				IF F_ChkSettingLimit(stControlSettingIn.nInputNumber, TO_LREAL(stControlSettingIn.fInputFloat), stSettings[nRowIndex], stInfo => stInfo) THEN
					IF stSettings[nRowIndex].eDataType = E_DataType.eDataType_bool THEN
						F_TrackSettingChangesB(stControlSettingIn.bInputBool, stSettings[nRowIndex], sChanges);
					ELSIF stSettings[nRowIndex].eDataType = E_DataType.eDataType_int THEN
						F_TrackSettingChangesI(stControlSettingIn.nInputNumber, stSettings[nRowIndex], sChanges);
					ELSIF stSettings[nRowIndex].eDataType = E_DataType.eDataType_lreal THEN
						F_TrackSettingChangesF(stControlSettingIn.fInputFloat, stSettings[nRowIndex], sChanges);
					ELSIF stSettings[nRowIndex].eDataType = E_DataType.eDataType_wstring THEN
						F_TrackSettingChangesWs(stControlSettingIn.wsInputString, stSettings[nRowIndex], sChanges);
					ELSIF stSettings[nRowIndex].eDataType = E_DataType.eDataType_time_ms THEN
						F_TrackSettingChangesT(TO_TIME(stControlSettingIn.nInputNumber), stSettings[nRowIndex], sChanges);
					ELSIF stSettings[nRowIndex].eDataType = E_DataType.eDataType_time_s THEN
						F_TrackSettingChangesT(TO_TIME((stControlSettingIn.fInputFloat) * 1000), stSettings[nRowIndex], sChanges);
					ELSIF stSettings[nRowIndex].eDataType = E_DataType.eDataType_time_m THEN
						F_TrackSettingChangesT(TO_TIME((stControlSettingIn.fInputFloat) * 60000), stSettings[nRowIndex], sChanges);
					ELSIF stSettings[nRowIndex].eDataType = E_DataType.eDataType_time_h THEN
						F_TrackSettingChangesT(TO_TIME((stControlSettingIn.fInputFloat) * 360000), stSettings[nRowIndex], sChanges);
					END_IF
				ELSE
					tofInfo.IN := TRUE;
				END_IF
				
			3: // min > user level admin
				IF (eUserLevel < E_User_Level.eUser_Level_Admin) 
					OR ((stSettings[nRowIndex].eUserLevel = E_User_Level.eUser_Level_Programmer) AND (eUserLevel <> E_User_Level.eUser_Level_Programmer))
				THEN
					tofInfo.IN :=	TRUE;
					stInfo.wsName := "incorrect user level";
					stInfo.wsNameId := "incorrectuserlevel";
				ELSE
					stSettings[nRowIndex].fValueMin := stControlSettingIn.fInputFloat;
				END_IF
				
			4: // max > user level admin
				IF (eUserLevel < E_User_Level.eUser_Level_Admin) 
					OR ((stSettings[nRowIndex].eUserLevel = E_User_Level.eUser_Level_Programmer) AND (eUserLevel <> E_User_Level.eUser_Level_Programmer))
				THEN
					tofInfo.IN :=	TRUE;
					stInfo.wsName := "incorrect user level";
					stInfo.wsNameId := "incorrectuserlevel";
				ELSE
					stSettings[nRowIndex].fValueMax := stControlSettingIn.fInputFloat;
				END_IF
				
			5: // unit only write by programmer
				;
					
			6: // user level admin
				IF (eUserLevel < E_User_Level.eUser_Level_Admin) 
					OR ((stSettings[nRowIndex].eUserLevel = E_User_Level.eUser_Level_Programmer) AND (eUserLevel <> E_User_Level.eUser_Level_Programmer))
				THEN
					tofInfo.IN :=	TRUE;
					stInfo.wsName := "incorrect user level";
					stInfo.wsNameId := "incorrectuserlevel";
				ELSE
					IF (stControlSettingIn.eUserLevel = E_User_Level.eUser_Level_Programmer) AND (eUserLevel < E_User_Level.eUser_Level_Programmer) THEN
						tofInfo.IN :=	TRUE;
						stInfo.wsName := "incorrect user level";
						stInfo.wsNameId := "incorrectuserlevel";						
					ELSE
						stSettings[nRowIndex].eUserLevel := stControlSettingIn.eUserLevel;
					END_IF	
				END_IF
				
			7: // type only write by programmer
				;
				
			8: // recipe level manager
				IF (eUserLevel < E_User_Level.eUser_Level_Manager) 
					OR ((stSettings[nRowIndex].eUserLevel = E_User_Level.eUser_Level_Programmer) AND (eUserLevel <> E_User_Level.eUser_Level_Programmer))
				THEN
					tofInfo.IN :=	TRUE;
					stInfo.wsName := "incorrect user level";
					stInfo.wsNameId := "incorrectuserlevel";
				ELSE
					stSettings[nRowIndex].eRecipeMode := stControlSettingIn.eRecipeMode;
				END_IF 				
		END_CASE
	END_IF
END_IF

tofInfo.PT := T#2S;
tofInfo();
tofInfo.IN := FALSE;
		
stControlSettingOut.bVisibleInfo := tofInfo.Q;
stControlSettingOut.stInfo := stInfo;

END_FUNCTION_BLOCK

// ---- POUs/System/Utilities/Functions/F_ColorToStringHexColor.TcPOU
FUNCTION F_ColorToStringHexColor : STRING
VAR_INPUT
	color : UDINT;
END_VAR

IF color = STATICS.stColor.None THEN
	F_ColorToStringHexColor := STATICS.stColor.NoneString;
ELSIF color = STATICS.stColor.Transparent THEN
	F_ColorToStringHexColor := STATICS.stColor.TransparentString;	
ELSIF color = STATICS.stColor.Theme THEN
	F_ColorToStringHexColor := STATICS.stColor.ThemeString;
ELSE
	F_ColorToStringHexColor  := Concat(
								'#',
								Delete(
									DWORD_TO_HEXSTR(
											color,
											8,
											FALSE)
									,2
									,1));//#hexadecimal
END_IF

END_FUNCTION

// ---- POUs/HMI/Utilities/Validation/F_ChkSettingUserLevel.TcPOU
FUNCTION F_ChkSettingUserLevel : BOOL
VAR_INPUT
	eLevel		: E_User_Level;
END_VAR
VAR_IN_OUT
	stSetting 	: ST_Data_Item;
END_VAR
VAR_OUTPUT
	stInfo 		: ST_Text;
END_VAR

F_ChkSettingUserLevel := FALSE;

IF (eUserLevel < stSetting.eUserLevel) THEN
	stInfo.wsName := "incorrect user level";
	stInfo.wsNameId := "incorrectuserlevel";
	RETURN;
END_IF

IF(stSetting.eDataType = E_DataType.eDataType_None)	THEN
	stInfo.wsName := "incorrect type";
	stInfo.wsNameId := "incorrecttype";
	RETURN;					
END_IF

F_ChkSettingUserLevel := TRUE;

END_FUNCTION

// ---- POUs/HMI/Utilities/Validation/F_ChkSettingLimit.TcPOU
FUNCTION F_ChkSettingLimit : BOOL
VAR_INPUT
	nValue		: INT;
	fValue		: LREAL;
END_VAR
VAR_IN_OUT
	stSetting 	: ST_Data_Item;
END_VAR
VAR_OUTPUT
	stInfo 		: ST_Text;
END_VAR

CASE stSetting.eDataType OF
	E_DataType.eDataType_int,
	E_DataType.eDataType_time_ms:
		F_ChkSettingLimit := F_ChkSettingLimitN(nValue, stSetting, stInfo => stInfo);
ELSE
		F_ChkSettingLimit := F_ChkSettingLimitF(fValue, stSetting, stInfo => stInfo);
END_CASE

END_FUNCTION

// ---- POUs/HMI/Utilities/Validation/F_ChkSettingLimitN.TcPOU
FUNCTION F_ChkSettingLimitN : BOOL
VAR_IN_OUT
	nValue		: INT;
	stSetting 	: ST_Data_Item;
END_VAR
VAR_OUTPUT
	stInfo 		: ST_Text;
END_VAR

F_ChkSettingLimitN := FALSE;

IF (stSetting.eDataType = E_DataType.eDataType_int) AND nValue > stSetting.fValueMax THEN
	stInfo.wsName := "input to high";
	stInfo.wsNameId := "inputtohigh";
	RETURN;
END_IF

IF (stSetting.eDataType = E_DataType.eDataType_int) AND nValue < stSetting.fValueMin THEN
	stInfo.wsName := "input to low";
	stInfo.wsNameId := "inputtolow";
	RETURN;
END_IF

IF (stSetting.eDataType = E_DataType.eDataType_time_ms) AND nValue > stSetting.fValueMax THEN
	stInfo.wsName := "input to high";
	stInfo.wsNameId := "inputtohigh";
	RETURN;
END_IF

IF (stSetting.eDataType = E_DataType.eDataType_time_ms) AND nValue < stSetting.fValueMin THEN
	stInfo.wsName := "input to low";
	stInfo.wsNameId := "inputtolow";
	RETURN;
END_IF

F_ChkSettingLimitN := TRUE;

END_FUNCTION

// ---- POUs/HMI/Utilities/Validation/F_ChkSettingLimitF.TcPOU
FUNCTION F_ChkSettingLimitF : BOOL
VAR_IN_OUT
	fValue		: LREAL;
	stSetting 	: ST_Data_Item;
END_VAR
VAR_OUTPUT
	stInfo 		: ST_Text;
END_VAR

F_ChkSettingLimitF := FALSE;

IF (stSetting.eDataType = E_DataType.eDataType_lreal) AND fValue > stSetting.fValueMax THEN
	stInfo.wsName := "input to high";
	stInfo.wsNameId := "inputtohigh";
	RETURN;
END_IF

IF (stSetting.eDataType = E_DataType.eDataType_lreal) AND fValue < stSetting.fValueMin THEN
	stInfo.wsName := "input to low";
	stInfo.wsNameId := "inputtolow";
	RETURN;
END_IF

IF (stSetting.eDataType = E_DataType.eDataType_time_s) AND fValue > stSetting.fValueMax THEN
	stInfo.wsName := "input to high";
	stInfo.wsNameId := "inputtohigh";
	RETURN;
END_IF

IF (stSetting.eDataType = E_DataType.eDataType_time_s) AND fValue < stSetting.fValueMin THEN
	stInfo.wsName := "input to low";
	stInfo.wsNameId := "inputtolow";
	RETURN;
END_IF

IF (stSetting.eDataType = E_DataType.eDataType_time_m) AND fValue > stSetting.fValueMax THEN
	stInfo.wsName := "input to high";
	stInfo.wsNameId := "inputtohigh";
	RETURN;
END_IF

IF (stSetting.eDataType = E_DataType.eDataType_time_m) AND fValue < stSetting.fValueMin THEN
	stInfo.wsName := "input to low";
	stInfo.wsNameId := "inputtolow";
	RETURN;
END_IF

IF (stSetting.eDataType = E_DataType.eDataType_time_h) AND fValue > stSetting.fValueMax THEN
	stInfo.wsName := "input to high";
	stInfo.wsNameId := "inputtohigh";
	RETURN;
END_IF

IF (stSetting.eDataType = E_DataType.eDataType_time_h) AND fValue < stSetting.fValueMin THEN
	stInfo.wsName := "input to low";
	stInfo.wsNameId := "inputtolow";
	RETURN;
END_IF

F_ChkSettingLimitF := TRUE;

END_FUNCTION

// ---- POUs/HMI/Utilities/Tracking/F_TrackSettingChangesB.TcPOU
FUNCTION F_TrackSettingChangesB : BOOL
VAR_INPUT
	bValue		: BOOL;
END_VAR
VAR_IN_OUT
	stSetting	: ST_Data_Item;
	sChanges	: STRING;
END_VAR

IF stSetting.bValue <> bValue THEN
	sChanges := Concat7(sChanges, '$N ', WSTRING_TO_STRING(stSetting.stName.wsName), ' ', TO_STRING(stSetting.bValue), ' -> ', TO_STRING(bValue));
END_IF

stSetting.bValue := bValue;
F_TrackSettingChangesB := TRUE;

END_FUNCTION

// ---- POUs/HMI/Utilities/Tracking/F_TrackSettingChangesI.TcPOU
FUNCTION F_TrackSettingChangesI : BOOL
VAR_INPUT
	nValue		: INT;
END_VAR
VAR_IN_OUT
	stSetting	: ST_Data_Item;
	sChanges	: STRING;
END_VAR

IF stSetting.nValue <> nValue THEN
	sChanges := Concat7(sChanges, '$N ', WSTRING_TO_STRING(stSetting.stName.wsName), ' ', TO_STRING(stSetting.nValue), ' -> ', TO_STRING(nValue));
END_IF

stSetting.nValue := nValue;
F_TrackSettingChangesI := TRUE;

END_FUNCTION

// ---- POUs/HMI/Utilities/Tracking/F_TrackSettingChangesF.TcPOU
FUNCTION F_TrackSettingChangesF : BOOL
VAR_INPUT
	fValue		: REAL;
END_VAR
VAR_IN_OUT
	stSetting	: ST_Data_Item;
	sChanges	: STRING;
END_VAR

IF stSetting.fValue <> fValue THEN
	sChanges := Concat7(sChanges, '$N ', WSTRING_TO_STRING(stSetting.stName.wsName), ' ', TO_STRING(stSetting.fValue), ' -> ', TO_STRING(fValue));
END_IF

stSetting.fValue := fValue;
F_TrackSettingChangesF := TRUE;

END_FUNCTION

// ---- POUs/HMI/Utilities/Tracking/F_TrackSettingChangesWs.TcPOU
FUNCTION F_TrackSettingChangesWs : BOOL
VAR_INPUT
	sValue		: WSTRING;
END_VAR
VAR_IN_OUT
	stSetting	: ST_Data_Item;
	sChanges	: STRING;
END_VAR

IF stSetting.sValue <> sValue THEN
	sChanges := Concat7(sChanges, '$N ', WSTRING_TO_STRING(stSetting.stName.wsName), ' ', TO_STRING(stSetting.sValue), ' -> ', TO_STRING(sValue));
END_IF

stSetting.sValue := sValue;
F_TrackSettingChangesWs := TRUE;

END_FUNCTION

// ---- POUs/HMI/Utilities/Tracking/F_TrackSettingChangesT.TcPOU
FUNCTION F_TrackSettingChangesT : BOOL
VAR_INPUT
	tValue		: TIME;
END_VAR
VAR_IN_OUT
	stSetting	: ST_Data_Item;
	sChanges	: STRING;
END_VAR

IF stSetting.tValue <> tValue THEN
	sChanges := Concat7(sChanges, '$N ', WSTRING_TO_STRING(stSetting.stName.wsName), ' ', TO_STRING(stSetting.tValue), ' -> ', TO_STRING(tValue));
END_IF

stSetting.tValue := tValue;
F_TrackSettingChangesT := TRUE;

END_FUNCTION

// ---- POUs/HMI/Utilities/FB_MonitoringHandling.TcPOU
FUNCTION_BLOCK FB_MonitoringHandling
VAR_INPUT
	nDigits				: INT; //number of digits after decimal point
END_VAR
VAR_IN_OUT
	stMonitoring		: ARRAY[*] OF ST_Data_Item;
	stMonitoringView	: ARRAY[*] OF ST_Data_Item_String;
END_VAR
VAR_OUTPUT
	
END_VAR
VAR
	ii, nLb, nUb		: DINT;
END_VAR

// clear MonitoringView
nLb := LOWER_BOUND(stMonitoringView, 1);
nUb := UPPER_BOUND(stMonitoringView, 1);
FOR ii := nLb TO nUb DO
	MEMSET(ADR(stMonitoringView[ii]), 0, SIZEOF(stMonitoringView[ii]));
END_FOR

// write MonitoringView
nLb := MAX(nLb, LOWER_BOUND(stMonitoring, 1));
nUb := MIN(nUb, UPPER_BOUND(stMonitoring, 1));
FOR ii := nLb TO nUb DO

	stMonitoringView[ii].stGroup := stMonitoring[ii].stGroup;
	stMonitoringView[ii].stName := stMonitoring[ii].stName;
	stMonitoringView[ii].stUnit := stMonitoring[ii].stUnit;
	
	IF (stMonitoring[ii].stName.wsName = "" AND stMonitoring[ii].stName.wsNameId = "") THEN
		stMonitoringView[ii].stDataType.wsName := stMonitoringView[ii].stDataType.wsNameId :="";	
	ELSIF stMonitoring[ii].eDataType = E_DataType.eDataType_None THEN
		stMonitoringView[ii].stDataType.wsName := stMonitoringView[ii].stDataType.wsNameId :="none";	
	ELSIF stMonitoring[ii].eDataType = E_DataType.eDataType_bool THEN
		stMonitoringView[ii].stDataType.wsName := stMonitoringView[ii].stDataType.wsNameId :="bool";
	ELSIF  stMonitoring[ii].eDataType = E_DataType.eDataType_int THEN
		stMonitoringView[ii].stDataType.wsName := stMonitoringView[ii].stDataType.wsNameId :="int";
	ELSIF  stMonitoring[ii].eDataType = E_DataType.eDataType_lreal THEN
		stMonitoringView[ii].stDataType.wsName := stMonitoringView[ii].stDataType.wsNameId :="lreal";
	ELSIF  stMonitoring[ii].eDataType = E_DataType.eDataType_time_ms THEN
		stMonitoringView[ii].stDataType.wsName := stMonitoringView[ii].stDataType.wsNameId :="time_ms";
	ELSIF  stMonitoring[ii].eDataType = E_DataType.eDataType_time_s THEN
		stMonitoringView[ii].stDataType.wsName := stMonitoringView[ii].stDataType.wsNameId :="time_s";		
	ELSIF  stMonitoring[ii].eDataType = E_DataType.eDataType_wstring THEN
		stMonitoringView[ii].stDataType.wsName := stMonitoringView[ii].stDataType.wsNameId :="wstring";
	END_IF
	
	IF (stMonitoring[ii].stName.wsName = "" AND stMonitoring[ii].stName.wsNameId = "") THEN
		stMonitoringView[ii].stValue.wsName := stMonitoringView[ii].stValue.wsNameId :="";
	ELSIF stMonitoring[ii].eDataType = E_DataType.eDataType_bool THEN
		IF stMonitoring[ii].bValue THEN
			stMonitoringView[ii].stValue.wsName := stMonitoringView[ii].stValue.wsNameId :="true";
		ELSE
			stMonitoringView[ii].stValue.wsName := stMonitoringView[ii].stValue.wsNameId :="false";
		END_IF
	ELSIF stMonitoring[ii].eDataType = E_DataType.eDataType_int THEN
		stMonitoringView[ii].stValue.wsName := TO_WSTRING(stMonitoring[ii].nValue);
	ELSIF stMonitoring[ii].eDataType = E_DataType.eDataType_lreal THEN
		stMonitoringView[ii].stValue.wsName := TO_WSTRING(LREAL_TO_FMTSTR(stMonitoring[ii].fValue,nDigits,FALSE));
	ELSIF stMonitoring[ii].eDataType = E_DataType.eDataType_wstring THEN
		stMonitoringView[ii].stValue.wsName := TO_WSTRING(stMonitoring[ii].sValue);
	ELSIF stMonitoring[ii].eDataType = E_DataType.eDataType_time_ms THEN
		stMonitoringView[ii].stValue.wsName := TO_WSTRING(stMonitoring[ii].tValue);
	END_IF
END_FOR

END_FUNCTION_BLOCK

// ---- POUs/System/Utilities/Functions/F_OR_REF.TcPOU
FUNCTION F_OR_REF : BOOL
VAR_IN_OUT
	bValueRoot		: BOOL;
END_VAR
VAR_INPUT
	bValueCombine	: BOOL;
END_VAR

bValueRoot := bValueRoot OR bValueCombine;

END_FUNCTION

// ---- POUs/Plant/P_Plant.TcPOU
PROGRAM P_Plant
VAR_INPUT	
	/// - stations, modules and components -
	aIStaton			: ARRAY[0..E_Station.eStation_nMaxIdx] OF IStation;
	aIModule			: ARRAY[0..E_Module.eModule_nMaxIdx] OF IModule;
	aIComponent			: ARRAY[0..E_Component.eComponent_nMaxIdx] OF ITFComponent;
END_VAR
VAR
	bInitSettingPlant		: BOOL;
	bInitSettingProduct		: BOOL;
	bInitSettingProduction	: BOOL;
	
	// plant empty... 
	bPlantEmptyActiv	: BOOL;
	bPlantEmpty			: BOOL;
	// logger, notification handler
	ILog				: I_Logger;
	IEvent				: I_EventHandler;
	
	/// private var's
	ii					: INT;
	b1stShot			: BOOL;
	tonDelay			: TON;
	
	/// clear text info
	aSClearText			: ARRAY[0..eLanguage_maxIdx] OF T_MaxString;
	bInitCounter		: BOOL;
	
	stSettingsPlantBackup		: ARRAY[0..E_PlantSettings.ePlantSetting_nMaxIdx] OF ST_Data_Item;
	stSettingsProductBackup		: ARRAY[0..E_ProductSettings.eProductSettings_nMaxIdx] OF ST_Data_Item;
	stSettingsProductionBackup	: ARRAY[0..E_ProductionSettings.eProductionSettings_nMaxIdx] OF ST_Data_Item;
END_VAR

///
/// Plant
///

// run 
aSClearText[EN] := 'Manage settings for plant, product and production';
M_SettingsPlant();
M_SettingsProduct();
M_SettingsProduction();

aSClearText[EN] := 'Calling modules...';
FOR ii := 0 TO E_Module.eModule_nMaxIdx DO
	IF aIModule[ii] = 0 THEN
		CONTINUE;
	END_IF
	
	aIModule[ii].EmergencyStopOk := P_Safety.EmergencyStopOk;
	aIModule[ii].M_Run(); // station run is called by its module
END_FOR

aSClearText[EN] := 'Calling stations, collect infos...';
b1stShot := TRUE;
FOR ii := 0 TO E_Station.eStation_nMaxIdx DO
	IF aIStaton[ii] = 0 THEN
		CONTINUE;
	END_IF
	
	F_AND_REF_EX(stGlobalModuleInfo.bStation_All_Auto, aIStaton[ii].OpMode = E_OpMode.eOpMode_auto, b1stShot);
	F_OR_REF_EX(stGlobalModuleInfo.bStation_Any_Step, aIStaton[ii].OpMode = E_OpMode.eOpMode_step, b1stShot);
	F_OR_REF_EX(stGlobalModuleInfo.bStation_Any_Manual, aIStaton[ii].OpMode = E_OpMode.eOpMode_manual, b1stShot);
	
	F_OR_REF_EX(stGlobalModuleInfo.bStation_Any_Error, aIStaton[ii].State = E_ComponentState.eComponentState_error, b1stShot);
	F_OR_REF_EX(stGlobalModuleInfo.bStation_Any_Warning, aIStaton[ii].State = E_ComponentState.eComponentState_warning, b1stShot);
	F_OR_REF_EX(stGlobalModuleInfo.bStation_Any_Info, aIStaton[ii].State = E_ComponentState.eComponentState_info, b1stShot);
	
	F_AND_REF_EX(stGlobalModuleInfo.bStation_All_Started, (aIStaton[ii].OpMode = E_OpMode.eOpMode_auto OR aIStaton[ii].OpMode = E_OpMode.eOpMode_step) AND aIStaton[ii].RunCycle, b1stShot);
	F_AND_REF_EX(stGlobalModuleInfo.bStation_All_Stopped, aIStaton[ii].Stopped, b1stShot);
	F_AND_REF_EX(stGlobalModuleInfo.bStation_All_InHome, aIStaton[ii].InHome, b1stShot);
	F_OR_REF_EX(stGlobalModuleInfo.bStation_Any_Homing, aIStaton[ii].Homing, b1stShot);
	
	b1stShot := FALSE;
END_FOR

aSClearText[EN] := 'Calling stations, plant components...';
FOR ii := 0 TO E_Component.eComponent_nMaxIdx DO
	IF aIComponent[ii] = 0 THEN
		CONTINUE;
	END_IF
	
	aIComponent[ii].Run();
END_FOR

aSClearText[EN] := 'Calling counter, check reset...';
IF HMI.stHmi.stIn.stMain.stButton_Reset.bClick THEN
	M_Reset();
END_IF

M_Counter();

IF bPlantEmptyActiv THEN
	IEvent.Select(Tc_Events.PlantEventClass.InfoEvent)
		  .ArgSetWString(CONST.stTextListGlobal.stText_emptymodeactive.wsName)
		  .Raise();
END_IF

{attribute 'monitoring' := 'call'}
PROPERTY PUBLIC CarrierColumnDistance : LREAL
GET
CarrierColumnDistance := stSettings.stProduct_Settings[E_ProductSettings.eProductSettings_CarrierColumnDistance].fValue;
END_GET
END_PROPERTY

{attribute 'monitoring' := 'call'}
PROPERTY PUBLIC CarrierCoordinateFirstWorkpieceX : LREAL
GET
CarrierCoordinateFirstWorkpieceX := stSettings.stProduct_Settings[E_ProductSettings.eProductSettings_CarrierCoordinateFirstWorkpieceX].fValue;
END_GET
END_PROPERTY

{attribute 'monitoring' := 'call'}
PROPERTY PUBLIC CarrierCoordinateFirstWorkpieceY : LREAL
GET
CarrierCoordinateFirstWorkpieceY := stSettings.stProduct_Settings[E_ProductSettings.eProductSettings_CarrierCoordinateFirstWorkpieceY].fValue;
END_GET
END_PROPERTY

{attribute 'monitoring' := 'call'}
PROPERTY PUBLIC CarrierDimensionX : LREAL
GET
CarrierDimensionX := stSettings.stProduct_Settings[E_ProductSettings.eProductSettings_CarrierDimensionX].fValue;
END_GET
END_PROPERTY

{attribute 'monitoring' := 'call'}
PROPERTY PUBLIC CarrierDimensionY : LREAL
GET
CarrierDimensionY := stSettings.stProduct_Settings[E_ProductSettings.eProductSettings_CarrierDimensionY].fValue;
END_GET
END_PROPERTY

{attribute 'monitoring' := 'call'}
PROPERTY PUBLIC CarrierInitialStatus : eTcaWorkpieceStatus
GET
CarrierInitialStatus := stSettings.stProduct_Settings[E_ProductSettings.eProductSettings_CarrierInitialStatus].nValue;
END_GET
END_PROPERTY

{attribute 'monitoring' := 'call'}
PROPERTY PUBLIC CarrierLayout : INT
GET
CarrierLayout := stSettings.stProduct_Settings[E_ProductSettings.eProductSettings_CarrierLayout].nValue;
END_GET
END_PROPERTY

{attribute 'monitoring' := 'call'}
PROPERTY PUBLIC CarrierPositionsInColumn : INT
GET
CarrierPositionsInColumn := stSettings.stProduct_Settings[E_ProductSettings.eProductSettings_CarrierPositionsInColumn].nValue;
END_GET
END_PROPERTY

{attribute 'monitoring' := 'call'}
PROPERTY PUBLIC CarrierPositionsInRow : INT
GET
CarrierPositionsInRow := stSettings.stProduct_Settings[E_ProductSettings.eProductSettings_CarrierPositionsInRow].nValue;
END_GET
END_PROPERTY

{attribute 'monitoring' := 'call'}
PROPERTY PUBLIC CarrierRequestStatus : eTcaWorkpieceStatus
GET
CarrierRequestStatus := stSettings.stProduct_Settings[E_ProductSettings.eProductSettings_CarrierRequestStatus].nValue;
END_GET
END_PROPERTY

{attribute 'monitoring' := 'call'}
PROPERTY PUBLIC CarrierRowDistance : LREAL
GET
CarrierRowDistance := stSettings.stProduct_Settings[E_ProductSettings.eProductSettings_CarrierRowDistance].fValue;
END_GET
END_PROPERTY

PROPERTY HeatingPlateEnable : BOOL
GET
HeatingPlateEnable := stSettings.stProduct_Settings[E_ProductSettings.eProductSettings_HeatingPlateEnable].bValue;
END_GET
END_PROPERTY

PROPERTY HeatingPlateTemperature : INT
GET
HeatingPlateTemperature := stSettings.stProduct_Settings[E_ProductSettings.eProductSettings_HeatingPlateTemperatur].nValue;
END_GET
END_PROPERTY

METHOD M_Counter : BOOL
VAR_INPUT
END_VAR
//init counter
IF NOT bInitCounter THEN
	bInitCounter := TRUE;
	
	FOR ii := 0 TO CONST.iMaxIdxCounter DO
		MEMSET(ADR(stCounter[ii].stGroup), 0, SIZEOF(stCounter[ii].stGroup));
		MEMSET(ADR(stCounter[ii].stName), 0, SIZEOF(stCounter[ii].stName));
		stCounter[ii].stGroup.wsNameId := stCounter[ii].stGroup.wsName := TO_WSTRING(ii);
	END_FOR
	
	stCounter[E_Counter.eCounter_General].stName.wsName := "Zaehler | Gesamt";
	//stCounter[E_Counter.eCounter_Maintenance].stName.wsName := "Zaehler | Wartung";
	stCounter[E_Counter.eCounter_Shift].stName.wsName := "Zaehler | Schicht";
	//stCounter[E_Counter.eCounter_Order].stName.wsName := "Zaehler | Auftrag";	
	//stCounter[E_Counter.eCounter_St001].stName.wsName := "Zaehler | St001_Eingabe_Takte";

	FOR ii := 0 TO CONST.iMaxIdxCounter DO
		stCounter[ii].stName.wsNameId := stCounter[ii].stName.wsName;
	END_FOR	
END_IF


FOR ii := 0 TO CONST.iMaxIdxCounter DO
	IF (stCounter[ii].eCurrentReactionOkLevel1 = E_CounterReaction.eCounterReaction_Info) THEN
		IEvent.Select(Tc_Events.PlantEventClass.InfoEvent)
			  .ArgSbInitWs(stTextListGlobal.stText_NG_Counter.wsName)
			  .ArgSbAppend(' | ')
			  .ArgSbAppendWs(stCounter[ii].stName.wsName)
			  .ArgSbAppendRaise(' | Level 1 Ok');
	END_IF
	IF (stCounter[ii].eCurrentReactionOkLevel2 = E_CounterReaction.eCounterReaction_Info) THEN
		IEvent.Select(Tc_Events.PlantEventClass.InfoEvent)
			  .ArgSbInitWs(stTextListGlobal.stText_NG_Counter.wsName)
			  .ArgSbAppend(' | ')
			  .ArgSbAppendWs(stCounter[ii].stName.wsName)
			  .ArgSbAppendRaise(' | Level 2 Ok');
	END_IF
	
	IF (stCounter[ii].eCurrentReactionOkLevel1 = E_CounterReaction.eCounterReaction_Warning) THEN
		IEvent.Select(Tc_Events.PlantEventClass.WarningEvent)
			  .ArgSbInitWs(stTextListGlobal.stText_NG_Counter.wsName)
			  .ArgSbAppend(' | ')
			  .ArgSbAppendWs(stCounter[ii].stName.wsName)
			  .ArgSbAppendRaise(' | Level 1 Ok');
	END_IF
	IF (stCounter[ii].eCurrentReactionOkLevel2 = E_CounterReaction.eCounterReaction_Warning) THEN
		IEvent.Select(Tc_Events.PlantEventClass.WarningEvent)
			  .ArgSbInitWs(stTextListGlobal.stText_NG_Counter.wsName)
			  .ArgSbAppend(' | ')
			  .ArgSbAppendWs(stCounter[ii].stName.wsName)
			  .ArgSbAppendRaise(' | Level 2 Ok');
	END_IF

	IF (stCounter[ii].eCurrentReactionOkLevel1 = E_CounterReaction.eCounterReaction_Error) THEN
		IEvent.Select(Tc_Events.PlantEventClass.ErrorEvent)
			  .ArgSbInitWs(stTextListGlobal.stText_NG_Counter.wsName)
			  .ArgSbAppend(' | ')
			  .ArgSbAppendWs(stCounter[ii].stName.wsName)
			  .ArgSbAppendRaise(' | Level 1 Ok');
	END_IF
	IF (stCounter[ii].eCurrentReactionOkLevel2 = E_CounterReaction.eCounterReaction_Error) THEN
		IEvent.Select(Tc_Events.PlantEventClass.ErrorEvent)
			  .ArgSbInitWs(stTextListGlobal.stText_NG_Counter.wsName)
			  .ArgSbAppend(' | ')
			  .ArgSbAppendWs(stCounter[ii].stName.wsName)
			  .ArgSbAppendRaise(' | Level 2 Ok');
	END_IF

	
	IF (stCounter[ii].eCurrentReactionNokLevel1 = E_CounterReaction.eCounterReaction_Info) THEN
		IEvent.Select(Tc_Events.PlantEventClass.InfoEvent)
			  .ArgSbInitWs(stTextListGlobal.stText_NG_Counter.wsName)
			  .ArgSbAppend(' | ')
			  .ArgSbAppendWs(stCounter[ii].stName.wsName)
			  .ArgSbAppendRaise(' | Level 1 NOk');
	END_IF
	IF (stCounter[ii].eCurrentReactionNokLevel2 = E_CounterReaction.eCounterReaction_Info) THEN
		IEvent.Select(Tc_Events.PlantEventClass.InfoEvent)
			  .ArgSbInitWs(stTextListGlobal.stText_NG_Counter.wsName)
			  .ArgSbAppend(' | ')
			  .ArgSbAppendWs(stCounter[ii].stName.wsName)
			  .ArgSbAppendRaise(' | Level 2 NOk');
	END_IF
	
	IF (stCounter[ii].eCurrentReactionNokLevel1 = E_CounterReaction.eCounterReaction_Warning) THEN
		IEvent.Select(Tc_Events.PlantEventClass.WarningEvent)
			  .ArgSbInitWs(stTextListGlobal.stText_NG_Counter.wsName)
			  .ArgSbAppend(' | ')
			  .ArgSbAppendWs(stCounter[ii].stName.wsName)
			  .ArgSbAppendRaise(' | Level 1 NOk');
	END_IF
	IF (stCounter[ii].eCurrentReactionNokLevel2 = E_CounterReaction.eCounterReaction_Warning) THEN
		IEvent.Select(Tc_Events.PlantEventClass.WarningEvent)
			  .ArgSbInitWs(stTextListGlobal.stText_NG_Counter.wsName)
			  .ArgSbAppend(' | ')
			  .ArgSbAppendWs(stCounter[ii].stName.wsName)
			  .ArgSbAppendRaise(' | Level 2 NOk');
	END_IF

	IF (stCounter[ii].eCurrentReactionNokLevel1 = E_CounterReaction.eCounterReaction_Error) THEN
		IEvent.Select(Tc_Events.PlantEventClass.ErrorEvent)
			  .ArgSbInitWs(stTextListGlobal.stText_NG_Counter.wsName)
			  .ArgSbAppend(' | ')
			  .ArgSbAppendWs(stCounter[ii].stName.wsName)
			  .ArgSbAppendRaise(' | Level 1 NOk');
	END_IF
	IF (stCounter[ii].eCurrentReactionNokLevel2 = E_CounterReaction.eCounterReaction_Error) THEN
		IEvent.Select(Tc_Events.PlantEventClass.ErrorEvent)
			  .ArgSbInitWs(stTextListGlobal.stText_NG_Counter.wsName)
			  .ArgSbAppend(' | ')
			  .ArgSbAppendWs(stCounter[ii].stName.wsName)
			  .ArgSbAppendRaise(' | Level 2 NOk');
	END_IF
	
	
	IF (stCounter[ii].eCurrentReactionTotalLevel1 = E_CounterReaction.eCounterReaction_Info) THEN
		IEvent.Select(Tc_Events.PlantEventClass.InfoEvent)
			  .ArgSbInitWs(stTextListGlobal.stText_NG_Counter.wsName)
			  .ArgSbAppend(' | ')
			  .ArgSbAppendWs(stCounter[ii].stName.wsName)
			  .ArgSbAppendRaise(' | Level 1 Total');
	END_IF
	IF (stCounter[ii].eCurrentReactionTotalLevel2 = E_CounterReaction.eCounterReaction_Info) THEN
		IEvent.Select(Tc_Events.PlantEventClass.InfoEvent)
			  .ArgSbInitWs(stTextListGlobal.stText_NG_Counter.wsName)
			  .ArgSbAppend(' | ')
			  .ArgSbAppendWs(stCounter[ii].stName.wsName)
			  .ArgSbAppendRaise(' | Level 2 Total');
	END_IF
	
	IF (stCounter[ii].eCurrentReactionTotalLevel1 = E_CounterReaction.eCounterReaction_Warning) THEN
		IEvent.Select(Tc_Events.PlantEventClass.WarningEvent)
			  .ArgSbInitWs(stTextListGlobal.stText_NG_Counter.wsName)
			  .ArgSbAppend(' | ')
			  .ArgSbAppendWs(stCounter[ii].stName.wsName)
			  .ArgSbAppendRaise(' | Level 1 Total');
	END_IF
	IF (stCounter[ii].eCurrentReactionTotalLevel2 = E_CounterReaction.eCounterReaction_Warning) THEN
		IEvent.Select(Tc_Events.PlantEventClass.WarningEvent)
			  .ArgSbInitWs(stTextListGlobal.stText_NG_Counter.wsName)
			  .ArgSbAppend(' | ')
			  .ArgSbAppendWs(stCounter[ii].stName.wsName)
			  .ArgSbAppendRaise(' | Level 2 Total');
	END_IF

	IF (stCounter[ii].eCurrentReactionTotalLevel1 = E_CounterReaction.eCounterReaction_Error) THEN
		IEvent.Select(Tc_Events.PlantEventClass.ErrorEvent)
			  .ArgSbInitWs(stTextListGlobal.stText_NG_Counter.wsName)
			  .ArgSbAppend(' | ')
			  .ArgSbAppendWs(stCounter[ii].stName.wsName)
			  .ArgSbAppendRaise(' | Level 1 Total');
	END_IF
	IF (stCounter[ii].eCurrentReactionTotalLevel2 = E_CounterReaction.eCounterReaction_Error) THEN
		IEvent.Select(Tc_Events.PlantEventClass.ErrorEvent)
			  .ArgSbInitWs(stTextListGlobal.stText_NG_Counter.wsName)
			  .ArgSbAppend(' | ')
			  .ArgSbAppendWs(stCounter[ii].stName.wsName)
			  .ArgSbAppendRaise(' | Level 2 Total');
	END_IF


	IF (stCounter[ii].eCurrentReactionNokLevel1 = E_CounterReaction.eCounterReaction_SerialFault_Warning) THEN
		IEvent.Select(Tc_Events.PlantEventClass.WarningEvent)
			  .ArgSbInitWs(stTextListGlobal.stText_NG_Counter.wsName)
			  .ArgSbAppend(' | ')
			  .ArgSbAppendWs(stCounter[ii].stName.wsName)
			  .ArgSbAppendRaise(' | Level 1 NOk Serienfehler');
	END_IF
	IF (stCounter[ii].eCurrentReactionNokLevel2 = E_CounterReaction.eCounterReaction_SerialFault_Warning) THEN
		IEvent.Select(Tc_Events.PlantEventClass.WarningEvent)
			  .ArgSbInitWs(stTextListGlobal.stText_NG_Counter.wsName)
			  .ArgSbAppend(' | ')
			  .ArgSbAppendWs(stCounter[ii].stName.wsName)
			  .ArgSbAppendRaise(' | Level 2 NOk Serienfehler');
	END_IF

	IF (stCounter[ii].eCurrentReactionNokLevel1 = E_CounterReaction.eCounterReaction_SerialFault_Error) THEN
		IEvent.Select(Tc_Events.PlantEventClass.ErrorEvent)
			  .ArgSbInitWs(stTextListGlobal.stText_NG_Counter.wsName)
			  .ArgSbAppend(' | ')
			  .ArgSbAppendWs(stCounter[ii].stName.wsName)
			  .ArgSbAppendRaise(' | Level 1 NOk Serienfehler');
	END_IF
	IF (stCounter[ii].eCurrentReactionNokLevel2 = E_CounterReaction.eCounterReaction_SerialFault_Error) THEN
		IEvent.Select(Tc_Events.PlantEventClass.ErrorEvent)
			  .ArgSbInitWs(stTextListGlobal.stText_NG_Counter.wsName)
			  .ArgSbAppend(' | ')
			  .ArgSbAppendWs(stCounter[ii].stName.wsName)
			  .ArgSbAppendRaise(' | Level 2 NOk Serienfehler');
	END_IF
END_FOR	

//reset counter

//rtrigResetCounter.CLK:=HMI.stRmthVisu.stVisuToPlc.bResetCounter;
//rtrigResetCounter();
//
//HMI.stRmthVisu.stVisuToPlc.iResetCounter:=LIMIT(1,HMI.stRmthVisu.stVisuToPlc.iResetCounter,(E_Counter.eCounter_Max-1));
//
//IF (HMI.stRmthVisu.stVisuToPlc.iResetCounter <=0) THEN
//	;
//ELSE
//	IF rtrigResetCounter.Q  AND bUserLevel[1] THEN
//		FOR ii:=2 TO (E_Counter.eCounter_Max-1) BY 1 DO 
//			IF(HMI.stRmthVisu.stVisuToPlc.iResetCounter = 1) THEN
//				F_Counter(E_CounterMode.eCounterMode_All_Clear,stCounter[ii]);	
//			END_IF		
//		END_FOR 
//		IF (HMI.stRmthVisu.stVisuToPlc.iResetCounter <> 1) THEN
//			F_Counter(E_CounterMode.eCounterMode_All_Clear,stCounter[LIMIT(2,HMI.stRmthVisu.stVisuToPlc.iResetCounter,(E_Counter.eCounter_Max-1))]);
//		END_IF
//	END_IF
//	//shift counter
//	IF HMI.stRmthVisu.stVisuToPlc.bResetShiftCounter  AND bUserLevel[E_User_Level.eUser_Level_Operator] THEN
//		F_Counter(E_CounterMode.eCounterMode_All_Clear,stCounter[E_Counter.eCounter_Shift]);
//	END_IF
//	bShiftCounter_Min:=FALSE;
//	bShiftCounter_Max:=FALSE;
//	HMI.stRmthVisu.stPlcToVisu.iResetShiftCounterCol:=Col.LightGray;
//	IF (stCounter[E_Counter.eCounter_Shift].fValue1 >= stCounter[E_Counter.eCounter_Shift].fValueMin) AND stCounter[E_Counter.eCounter_Shift].bYesNo THEN
//		P_Hmi.SetNotificationPrio(E_Notification.eNotification_Counter_Info, F_TranslateAndConcat2Txts("Info | Schichtzähler", ""), E_Priority.ePriority_info);
//		bShiftCounter_Min:=TRUE;
//		HMI.stRmthVisu.stPlcToVisu.iResetShiftCounterCol:=Col.LightBlue;
//	END_IF
//	IF (stCounter[E_Counter.eCounter_Shift].fValue1 >= stCounter[E_Counter.eCounter_Shift].fValueMax) AND stCounter[E_Counter.eCounter_Shift].bYesNo THEN
//		P_Hmi.SetNotificationPrio(E_Notification.eNotification_Counter_Warning, F_TranslateAndConcat2Txts("Warning | Schichtzähler", ""), E_Priority.ePriority_warning);
//		bShiftCounter_Max:=TRUE;
//		HMI.stRmthVisu.stPlcToVisu.iResetShiftCounterCol:=Col.Orange;
//	END_IF
//END_IF
//
END_METHOD

METHOD INTERNAL M_Init : BOOL
VAR_INPUT
END_VAR
// init components stuff here...
ILog := Services.ILog;
IEvent := Services.fbEventHandler;

bInitSettingPlant := FALSE;
bInitSettingProduct := FALSE;
bInitSettingProduction := FALSE;

aSClearText[EN] := 'Plant init done.';
M_Init := TRUE;
END_METHOD

METHOD INTERNAL M_RegisterComponent : BOOL
VAR_INPUT
	IComponent : ITFComponent;
END_VAR
aIComponent[IComponent.ID] := IComponent;
M_RegisterComponent := TRUE;
END_METHOD

METHOD INTERNAL M_RegisterModule : BOOL
VAR_INPUT
	IMod : IModule;
END_VAR
aIModule[IMod.Module] := IMod;
M_RegisterModule := TRUE;
END_METHOD

METHOD INTERNAL M_RegisterStation : BOOL
VAR_INPUT
	Ist : IStation;
END_VAR
aIStaton[ISt.Station] := ISt;
M_RegisterStation := TRUE;
END_METHOD

/// resets all additional components
METHOD M_Reset
VAR
END_VAR
// reset all additional components

//reset serial fault counter
FOR ii := 0 TO CONST.iMaxIdxCounter DO
	IF (stCounter[ii].eCurrentReactionNokLevel1 = E_CounterReaction.eCounterReaction_SerialFault_Warning) 
		OR (stCounter[ii].eCurrentReactionNokLevel1 = E_CounterReaction.eCounterReaction_SerialFault_Error)
		OR (stCounter[ii].eCurrentReactionNokLevel2 = E_CounterReaction.eCounterReaction_SerialFault_Warning) 
		OR (stCounter[ii].eCurrentReactionNokLevel2 = E_CounterReaction.eCounterReaction_SerialFault_Error)  
	THEN
		F_Counter(E_CounterMode.eCounterMode_SerialError_Clear, stCounter[ii]);
	END_IF
END_FOR
END_METHOD

METHOD M_SettingsPlant : BOOL
VAR_INPUT
END_VAR
// plant settings
IF NOT bInitSettingPlant THEN
	bInitSettingPlant := TRUE;
	stSettingsPlantBackup := stSettings.stPlant_Settings; // backup
	MEMSET(ADR(stSettings.stPlant_Settings), 0, SIZEOF(stSettings.stPlant_Settings)); // reset
	
	F_InitDynDataItem(E_PlantSettings.ePlantSetting_RecipeName, 		// settings index
		TO_WSTRING(E_PlantSettings.ePlantSetting_RecipeName),			// settings wsIndex
		CONST.stEmptyText,												// group
		stTextListGlobal.stText_RecipeName,								// name
		stTextListGlobal.stText_name, E_DataType.eDataType_wstring,		// unit & data type
		0, 0, 6,														// min, max & user level
		E_RecipeMode.eRecipeMode_ToFrom,														
		stSettings.stPlant_Settings);
		
	F_InitDynDataItem(E_PlantSettings.ePlantSetting_RecipeComment,
		TO_WSTRING(E_PlantSettings.ePlantSetting_RecipeComment),
		CONST.stEmptyText,
		stTextListGlobal.stText_RecipeComment,
		stTextListGlobal.stText_name, E_DataType.eDataType_wstring,
		0, 0, 6,
		E_RecipeMode.eRecipeMode_ToFrom,
		stSettings.stPlant_Settings);
		
	F_InitDynDataItem(E_PlantSettings.ePlantSetting_PlantName,
		TO_WSTRING(E_PlantSettings.ePlantSetting_PlantName),
		CONST.stEmptyText,
		stTextListGlobal.stText_PlantName,
		stTextListGlobal.stText_name, E_DataType.eDataType_wstring,
		0, 0, 6,
		E_RecipeMode.eRecipeMode_ToFrom,
		stSettings.stPlant_Settings);

	F_InitDynDataItem(E_PlantSettings.ePlantSetting_PlantNumber,
		TO_WSTRING(E_PlantSettings.ePlantSetting_PlantNumber),
		CONST.stEmptyText,
		stTextListGlobal.stText_PlantNumber,
		stTextListGlobal.stText_n, E_DataType.eDataType_int,
		0, 100000, 6,
		E_RecipeMode.eRecipeMode_ToFrom,
		stSettings.stPlant_Settings);

	F_RestoreSettingValues(stSettings.stPlant_Settings, stSettingsPlantBackup); // restore values
END_IF

// settings management
//F_Settings_Management(stSettings.stPlant_Settings);
END_METHOD

METHOD M_SettingsProduct : BOOL
VAR_INPUT
END_VAR
//init product settings
IF NOT bInitSettingProduct THEN
	bInitSettingProduct:=TRUE;
	stSettingsProductBackup := stSettings.stProduct_Settings; // backup
	MEMSET(ADR(stSettings.stProduct_Settings), 0, SIZEOF(stSettings.stProduct_Settings)); // reset

	F_InitDynDataItem(E_ProductSettings.eProductSettings_ProductNumber,	// settings index
		TO_WSTRING(E_ProductSettings.eProductSettings_ProductNumber),	// settings wsIndex
		F_CreateDynTextDefault("settingsproduct"),						// group
		stTextListGlobal.stText_RecipeName,								// name
		stTextListGlobal.stText_text, E_DataType.eDataType_wstring,		// unit & data type
		0, 100000000, 6,												// min, max & user level
		E_RecipeMode.eRecipeMode_ToFrom,
		stSettings.stProduct_Settings);		
	F_InitDynDataItem(E_ProductSettings.eProductSettings_ProductName,
		TO_WSTRING(E_ProductSettings.eProductSettings_ProductName),
		F_CreateDynTextDefault("settingsproduct"),
		F_CreateDynTextDefault("name"),
		stTextListGlobal.stText_text, E_DataType.eDataType_wstring,
		0, 0, 6,
		E_RecipeMode.eRecipeMode_ToFrom,
		stSettings.stProduct_Settings);		
	F_InitDynDataItem(E_ProductSettings.eProductSettings_ProductType,
		TO_WSTRING(E_ProductSettings.eProductSettings_ProductType),
		F_CreateDynTextDefault("settingsproduct"),
		F_CreateDynTextDefault("type"),
		stTextListGlobal.stText_n, E_DataType.eDataType_int,
		0, 10, 6,
		E_RecipeMode.eRecipeMode_ToFrom,
		stSettings.stProduct_Settings);		

	F_InitDynDataItem(E_ProductSettings.eProductSettings_TrolleyNumberOfCarriers,
		TO_WSTRING(E_ProductSettings.eProductSettings_TrolleyNumberOfCarriers),
		F_CreateDynTextDefault("settingsTrolley"),
		F_CreateDynTextDefault("Palettenanzahl"),
		stTextListGlobal.stText_n, E_DataType.eDataType_int,
		0, 50, 6,
		E_RecipeMode.eRecipeMode_ToFrom,
		stSettings.stProduct_Settings);		
	F_InitDynDataItem(E_ProductSettings.eProductSettings_TrolleyRackOriginX,
		TO_WSTRING(E_ProductSettings.eProductSettings_TrolleyRackOriginX),
		F_CreateDynTextDefault("settingsTrolley"),
		F_CreateDynTextDefault("Origin_X"),
		stTextListGlobal.stText_mm, E_DataType.eDataType_lreal,
		0, 1000, 6,
		E_RecipeMode.eRecipeMode_ToFrom,
		stSettings.stProduct_Settings);
	F_InitDynDataItem(E_ProductSettings.eProductSettings_TrolleyRackOriginY,
		TO_WSTRING(E_ProductSettings.eProductSettings_TrolleyRackOriginY),
		F_CreateDynTextDefault("settingsTrolley"),
		F_CreateDynTextDefault("Origin_Y"),
		stTextListGlobal.stText_mm, E_DataType.eDataType_lreal,
		0, 2000, 6,
		E_RecipeMode.eRecipeMode_ToFrom,
		stSettings.stProduct_Settings);		
	F_InitDynDataItem(E_ProductSettings.eProductSettings_TrolleyRackDivision,
		TO_WSTRING(E_ProductSettings.eProductSettings_TrolleyRackDivision),
		F_CreateDynTextDefault("settingsTrolley"),
		F_CreateDynTextDefault("Division"),
		stTextListGlobal.stText_mm, E_DataType.eDataType_lreal,
		0, 500, 6,
		E_RecipeMode.eRecipeMode_ToFrom,
		stSettings.stProduct_Settings);		
	F_InitDynDataItem(E_ProductSettings.eProductSettings_TrolleyCarrierDistance,
		TO_WSTRING(E_ProductSettings.eProductSettings_TrolleyCarrierDistance),
		F_CreateDynTextDefault("settingsTrolley"),
		F_CreateDynTextDefault("CarrierDistance"),
		stTextListGlobal.stText_mm, E_DataType.eDataType_lreal,
		0, 200, 6,
		E_RecipeMode.eRecipeMode_ToFrom,
		stSettings.stProduct_Settings);				
	
	F_InitDynDataItem(E_ProductSettings.eProductSettings_CarrierLayout,
		TO_WSTRING(E_ProductSettings.eProductSettings_CarrierLayout),
		F_CreateDynTextDefault("settingsCarrier"),
		F_CreateDynTextDefault("Layout"),
		stTextListGlobal.stText_n, E_DataType.eDataType_int,
		0, 6, 6,
		E_RecipeMode.eRecipeMode_ToFrom,
		stSettings.stProduct_Settings);		
	F_InitDynDataItem(E_ProductSettings.eProductSettings_CarrierDimensionX,
		TO_WSTRING(E_ProductSettings.eProductSettings_CarrierDimensionX),
		F_CreateDynTextDefault("settingsCarrier"),
		F_CreateDynTextDefault("DimensionX"),
		stTextListGlobal.stText_mm, E_DataType.eDataType_lreal,
		0, 600, 6,
		E_RecipeMode.eRecipeMode_ToFrom,
		stSettings.stProduct_Settings);	
	F_InitDynDataItem(E_ProductSettings.eProductSettings_CarrierDimensionY,
		TO_WSTRING(E_ProductSettings.eProductSettings_CarrierDimensionY),
		F_CreateDynTextDefault("settingsCarrier"),
		F_CreateDynTextDefault("DimensionY"),
		stTextListGlobal.stText_mm, E_DataType.eDataType_lreal,
		0, 600, 6,
		E_RecipeMode.eRecipeMode_ToFrom,
		stSettings.stProduct_Settings);	
	F_InitDynDataItem(E_ProductSettings.eProductSettings_CarrierRowDistance,
		TO_WSTRING(E_ProductSettings.eProductSettings_CarrierRowDistance),
		F_CreateDynTextDefault("settingsCarrier"),
		F_CreateDynTextDefault("RowDistance"),
		stTextListGlobal.stText_mm, E_DataType.eDataType_lreal,
		0, 600, 6,
		E_RecipeMode.eRecipeMode_ToFrom,
		stSettings.stProduct_Settings);	
	F_InitDynDataItem(E_ProductSettings.eProductSettings_CarrierColumnDistance,
		TO_WSTRING(E_ProductSettings.eProductSettings_CarrierColumnDistance),
		F_CreateDynTextDefault("settingsCarrier"),
		F_CreateDynTextDefault("ColumnDistance"),
		stTextListGlobal.stText_mm, E_DataType.eDataType_lreal,
		0, 600, 6,
		E_RecipeMode.eRecipeMode_ToFrom,
		stSettings.stProduct_Settings);	
	F_InitDynDataItem(E_ProductSettings.eProductSettings_CarrierPositionsInRow,
		TO_WSTRING(E_ProductSettings.eProductSettings_CarrierPositionsInRow),
		F_CreateDynTextDefault("settingsCarrier"),
		F_CreateDynTextDefault("PositionsInRow"),
		stTextListGlobal.stText_n, E_DataType.eDataType_int,
		0, 17, 6,
		E_RecipeMode.eRecipeMode_ToFrom,
		stSettings.stProduct_Settings);		
	F_InitDynDataItem(E_ProductSettings.eProductSettings_CarrierPositionsInColumn,
		TO_WSTRING(E_ProductSettings.eProductSettings_CarrierPositionsInColumn),
		F_CreateDynTextDefault("settingsCarrier"),
		F_CreateDynTextDefault("PositionsInColumn"),
		stTextListGlobal.stText_n, E_DataType.eDataType_int,
		0, 17, 6,
		E_RecipeMode.eRecipeMode_ToFrom,
		stSettings.stProduct_Settings);		
	F_InitDynDataItem(E_ProductSettings.eProductSettings_CarrierCoordinateFirstWorkpieceX,
		TO_WSTRING(E_ProductSettings.eProductSettings_CarrierCoordinateFirstWorkpieceX),
		F_CreateDynTextDefault("settingsCarrier"),
		F_CreateDynTextDefault("CoordinateFirstWorkpieceX"),
		stTextListGlobal.stText_mm, E_DataType.eDataType_lreal,
		0, 600, 6,
		E_RecipeMode.eRecipeMode_ToFrom,
		stSettings.stProduct_Settings);	
	F_InitDynDataItem(E_ProductSettings.eProductSettings_CarrierCoordinateFirstWorkpieceY,
		TO_WSTRING(E_ProductSettings.eProductSettings_CarrierCoordinateFirstWorkpieceY),
		F_CreateDynTextDefault("settingsCarrier"),
		F_CreateDynTextDefault("CoordinateFirstWorkpieceY"),
		stTextListGlobal.stText_mm, E_DataType.eDataType_lreal,
		0, 600, 6,
		E_RecipeMode.eRecipeMode_ToFrom,
		stSettings.stProduct_Settings);	
	F_InitDynDataItem(E_ProductSettings.eProductSettings_CarrierRequestStatus,
		TO_WSTRING(E_ProductSettings.eProductSettings_CarrierRequestStatus),
		F_CreateDynTextDefault("settingsCarrier"),
		F_CreateDynTextDefault("RequestStatus"),
		stTextListGlobal.stText_n, E_DataType.eDataType_int,
		0, 5, 6,
		E_RecipeMode.eRecipeMode_ToFrom,
		stSettings.stProduct_Settings);		
	F_InitDynDataItem(E_ProductSettings.eProductSettings_CarrierInitialStatus,
		TO_WSTRING(E_ProductSettings.eProductSettings_CarrierInitialStatus),
		F_CreateDynTextDefault("settingsCarrier"),
		F_CreateDynTextDefault("InitialStatus"),
		stTextListGlobal.stText_n, E_DataType.eDataType_int,
		0, 5, 6,
		E_RecipeMode.eRecipeMode_ToFrom,
		stSettings.stProduct_Settings);		
		
	F_InitDynDataItem(E_ProductSettings.eProductSettings_HeatingPlateEnable,
		TO_WSTRING(E_ProductSettings.eProductSettings_HeatingPlateEnable),
		F_CreateDynTextDefault("settingsHeatingPlate"),
		F_CreateDynTextDefault("Enable"),
		stTextListGlobal.stText_n, E_DataType.eDataType_bool,
		0, 5, 6,
		E_RecipeMode.eRecipeMode_ToFrom,
		stSettings.stProduct_Settings);		
	F_InitDynDataItem(E_ProductSettings.eProductSettings_HeatingPlateTemperatur,
		TO_WSTRING(E_ProductSettings.eProductSettings_HeatingPlateTemperatur),
		F_CreateDynTextDefault("settingsHeatingPlate"),
		F_CreateDynTextDefault("Temperature"),
		stTextListGlobal.stText_n, E_DataType.eDataType_int,
		0, 5, 6,
		E_RecipeMode.eRecipeMode_ToFrom,
		stSettings.stProduct_Settings);		



F_RestoreSettingValues(stSettings.stProduct_Settings, stSettingsProductBackup); // restore values
END_IF

// settings management
F_Settings_Management(stSettings.stProduct_Settings);

stSettings.stCarrier.ColumnDistance := CarrierColumnDistance;
stSettings.stCarrier.CoordinateFirstWorkpiece.fX := CarrierCoordinateFirstWorkpieceX;
stSettings.stCarrier.CoordinateFirstWorkpiece.fY := CarrierCoordinateFirstWorkpieceY;
stSettings.stCarrier.Dimension.fX := CarrierDimensionX;
stSettings.stCarrier.Dimension.fY := CarrierDimensionY;
stSettings.stCarrier.InitialStatus := CarrierInitialStatus;
stSettings.stCarrier.Layout := CarrierLayout;
stSettings.stCarrier.PositionsInColumn := CarrierPositionsInColumn;
stSettings.stCarrier.PositionsInRow := CarrierPositionsInRow;
stSettings.stCarrier.RequestStatus := CarrierRequestStatus;
stSettings.stCarrier.RowDistance := CarrierRowDistance;

stSettings.stTrolley.CarrierConfig := stSettings.stCarrier;
stSettings.stTrolley.CarrierDistance := TrolleyCarrierDistance;
stSettings.stTrolley.NumberOfCarriers := TrolleyNumberOfCarriers;
stSettings.stTrolley.RackDivision := TrolleyRackDivision;
stSettings.stTrolley.RackOrigin.fX := TrolleyRackOriginX;
stSettings.stTrolley.RackOrigin.fY := TrolleyRackOriginY;
stSettings.stTrolley.RackOrigin.fZ := TrolleyRackOriginZ;
END_METHOD

METHOD M_SettingsProduction : BOOL
VAR
END_VAR
// init  production settings
IF NOT bInitSettingProduction THEN
	bInitSettingProduction := TRUE;
	stSettingsProductionBackup := stSettings.stProduction_Settings; // backup
	MEMSET(ADR(stSettings.stProduction_Settings), 0, SIZEOF(stSettings.stProduction_Settings));		// reset

	F_InitDynDataItem(E_ProductionSettings.eProductionSettings_Override,	// settings index
		TO_WSTRING(E_ProductionSettings.eProductionSettings_Override),		// settings wsIndex
		F_CreateDynText("settingsproduction", 0),							// group
		stTextListGlobal.stText_PlantSpeedOverride,							// name
		stTextListGlobal.stText_percent, E_DataType.eDataType_int,			// unit & data type
		0, 1500, 6,															// min, max & user level
		E_RecipeMode.eRecipeMode_ToFrom,
		stSettings.stProduction_Settings);
		
	F_InitDynDataItem(E_ProductionSettings.eProductionSettings_OrderNumber,
		TO_WSTRING(E_ProductionSettings.eProductionSettings_OrderNumber),
		F_CreateDynText("settingsproduction", 0),
		stTextListGlobal.stText_OrderNumber,
		stTextListGlobal.stText_text, E_DataType.eDataType_wstring,
		0, 40, 6,
		E_RecipeMode.eRecipeMode_ToFrom,
		stSettings.stProduction_Settings);
		
	F_RestoreSettingValues(stSettings.stProduction_Settings, stSettingsProductionBackup); // restore values
END_IF

// settings management
F_Settings_Management(stSettings.stProduction_Settings);
END_METHOD

{attribute 'monitoring' := 'call'}
PROPERTY PUBLIC TrolleyCarrierDistance : LREAL
GET
TrolleyCarrierDistance := stSettings.stProduct_Settings[E_ProductSettings.eProductSettings_TrolleyCarrierDistance].fValue;
END_GET
END_PROPERTY

{attribute 'monitoring' := 'call'}
PROPERTY PUBLIC TrolleyNumberOfCarriers : INT
GET
TrolleyNumberOfCarriers := stSettings.stProduct_Settings[E_ProductSettings.eProductSettings_TrolleyNumberOfCarriers].nValue;
END_GET
END_PROPERTY

{attribute 'monitoring' := 'call'}
PROPERTY PUBLIC TrolleyRackDivision : LREAL
GET
TrolleyRackDivision := stSettings.stProduct_Settings[E_ProductSettings.eProductSettings_TrolleyRackDivision].fValue;
END_GET
END_PROPERTY

{attribute 'monitoring' := 'call'}
PROPERTY PUBLIC TrolleyRackOriginX : LREAL
GET
TrolleyRackOriginX := stSettings.stProduct_Settings[E_ProductSettings.eProductSettings_TrolleyRackOriginX].fValue;
END_GET
END_PROPERTY

{attribute 'monitoring' := 'call'}
PROPERTY PUBLIC TrolleyRackOriginY : LREAL
GET
TrolleyRackOriginY := stSettings.stProduct_Settings[E_ProductSettings.eProductSettings_TrolleyRackOriginY].fValue;
END_GET
END_PROPERTY

{attribute 'monitoring' := 'call'}
PROPERTY PUBLIC TrolleyRackOriginZ : LREAL
GET
TrolleyRackOriginZ := stSettings.stProduct_Settings[E_ProductSettings.eProductSettings_TrolleyRackOriginZ].fValue;
END_GET
END_PROPERTY

END_PROGRAM

// ---- POUs/System/Utilities/Functions/F_AND_REF_EX.TcPOU
FUNCTION F_AND_REF_EX : BOOL
VAR_IN_OUT
	bValueRoot		: BOOL;	
END_VAR
VAR_INPUT
	bValueCombine	: BOOL;
	bInitialize		: BOOL;
END_VAR

IF bInitialize THEN
	bValueRoot := TRUE;
END_IF
	
F_AND_REF(bValueRoot, bValueCombine);

END_FUNCTION

// ---- POUs/System/Utilities/Functions/F_AND_REF.TcPOU
FUNCTION F_AND_REF : BOOL
VAR_IN_OUT
	bValueRoot		: BOOL;
END_VAR
VAR_INPUT
	bValueCombine	: BOOL;
END_VAR

bValueRoot := bValueRoot AND bValueCombine;

END_FUNCTION

// ---- POUs/System/Utilities/Functions/F_OR_REF_EX.TcPOU
FUNCTION F_OR_REF_EX : BOOL
VAR_IN_OUT
	bValueRoot		: BOOL;	
END_VAR
VAR_INPUT
	bValueCombine	: BOOL;
	bInitialize		: BOOL;
END_VAR

IF bInitialize THEN
	bValueRoot := FALSE;
END_IF

F_OR_REF(bValueRoot, bValueCombine);

END_FUNCTION

// ---- POUs/System/Utilities/Counter/F_Counter.TcPOU
FUNCTION F_Counter : BOOL

VAR_INPUT
	eCounterMode : E_CounterMode;
END_VAR
VAR_IN_OUT
	stCounter	: ST_Counter_Item;//ST_Conunter;
END_VAR
VAR
END_VAR

IF (eCounterMode = E_CounterMode.eCounterMode_Ok_Up) THEN
	stCounter.nValueOk:=stCounter.nValueOk+1;
	stCounter.nValueSerialError:=0;
ELSIF (eCounterMode = E_CounterMode.eCounterMode_Ok_Down) THEN	
	stCounter.nValueOk:=stCounter.nValueOk-1;
ELSIF (eCounterMode = E_CounterMode.eCounterMode_Ok_Clear) THEN	
	stCounter.nValueOk:=0;		
ELSIF (eCounterMode = E_CounterMode.eCounterMode_Nok_Up) THEN	
	stCounter.nValueNok:=stCounter.nValueNok+1;	
	stCounter.nValueSerialError:=stCounter.nValueSerialError+1;
ELSIF (eCounterMode = E_CounterMode.eCounterMode_Nok_Down) THEN	
	stCounter.nValueNok:=stCounter.nValueNok-1;	
ELSIF (eCounterMode = E_CounterMode.eCounterMode_Nok_Clear) THEN	
	stCounter.nValueNok:=0;	
ELSIF (eCounterMode = E_CounterMode.eCounterMode_SerialError_Clear) THEN	
	stCounter.nValueSerialError:=0;		
ELSIF (eCounterMode = E_CounterMode.eCounterMode_All_Clear) THEN	
	stCounter.nValueOk:=0;
	stCounter.nValueNok:=0;
	stCounter.nValueSerialError:=0;			
END_IF

END_FUNCTION

// ---- POUs/System/Utilities/Functions/F_InitDynDataItem.TcPOU
FUNCTION F_InitDynDataItem : BOOL
VAR_INPUT
	nIndex				: INT;
	wsIndex				: WSTRING;
	stGroup				: ST_Text;
	stTitle				: ST_Text;
	stUnit				: ST_Text;	
	eDataType			: E_DataType;	
	fValueMin			: REAL;
	fValueMax			: REAL;
	// required user level, 0 = none
	nRequiredUserLevel	: INT := 0;	
	eRecipeMode			: E_RecipeMode;
END_VAR
VAR_IN_OUT
	astItems			: ARRAY[*] OF ST_Data_Item;
END_VAR
VAR
	nLb, nUb : INT;
END_VAR

nLb := TO_INT(LOWER_BOUND(astItems, 1));
nUb := TO_INT(UPPER_BOUND(astItems, 1));

// chk
IF nIndex < nLb OR nIndex > nUb THEN
	RETURN;
END_IF

astItems[nIndex].stIndex.nNameId := nIndex;
astItems[nIndex].stIndex.wsNameId := wsIndex;
astItems[nIndex].stIndex.wsName := wsIndex;

astItems[nIndex].stGroup := stGroup;
astItems[nIndex].stName := stTitle;

astItems[nIndex].eDataType := eDataType;
astItems[nIndex].fValueMin := fValueMin;
astItems[nIndex].fValueMax := fValueMax;
astItems[nIndex].stUnit := stUnit;

astItems[nIndex].eUserLevel := nRequiredUserLevel;

astItems[nIndex].eRecipeMode := eRecipeMode;

F_InitDynDataItem := TRUE;

END_FUNCTION

// ---- POUs/System/Utilities/Functions/F_RestoreSettingValues.TcPOU
FUNCTION F_RestoreSettingValues : BOOL
VAR_IN_OUT
	astSettings	: ARRAY[*] OF ST_Data_Item;
	astBackup	: ARRAY[*] OF ST_Data_Item;
END_VAR
VAR
	xx, nLb, nUb : INT;
	stItmTemp	 : REFERENCE TO ST_Data_Item;
END_VAR

nLb := TO_INT(LOWER_BOUND(astSettings, 1));
nUb := TO_INT(UPPER_BOUND(astSettings, 1));

FOR xx := nLb TO nUb DO 
	stItmTemp REF= F_FindBackupItem(astSettings[xx], astBackup);	// get backup
	F_CopyDataItemValues(astSettings[xx], stItmTemp);				// restore values	
END_FOR

F_RestoreSettingValues := TRUE;

END_FUNCTION

// ---- POUs/System/Utilities/Functions/F_FindBackupItem.TcPOU
FUNCTION F_FindBackupItem : REFERENCE TO ST_Data_Item
VAR_IN_OUT
	stItem		: ST_Data_Item;
	astBackup	: ARRAY[*] OF ST_Data_Item;
END_VAR
VAR
	xx, nLb, nUb	: INT;
	stEmpty			: ST_Data_Item;
END_VAR

nLb := TO_INT(LOWER_BOUND(astBackup, 1));
nUb := TO_INT(UPPER_BOUND(astBackup, 1));

// try to find item by wsNameId (in order to support insert and delete items)
IF stItem.stName.wsName <> CONST.wsEmpty THEN
	FOR xx := nLb TO nUb DO
		IF astBackup[xx].stIndex.wsNameId = stItem.stIndex.wsNameId THEN
			F_FindBackupItem REF= astBackup[xx]; // found, return
			RETURN;
		END_IF
	END_FOR
END_IF

// if not found, return item by index
IF stItem.stIndex.nNameId >= nLb AND stItem.stIndex.nNameId <= nUb THEN
	F_FindBackupItem REF= astBackup[stItem.stIndex.nNameId]; // found, return
	RETURN;
END_IF


// not found at all
F_FindBackupItem REF= stEmpty;

END_FUNCTION

// ---- POUs/System/Utilities/Functions/F_CopyDataItemValues.TcPOU
FUNCTION F_CopyDataItemValues : BOOL
VAR_IN_OUT
	stDst : ST_Data_Item;
	stSrc : ST_Data_Item;
END_VAR

stDst.bValue := stSrc.bValue;
stDst.tValue := stSrc.tValue;
stDst.sValue := stSrc.sValue;
stDst.nValue := stSrc.nValue;
stDst.fValue := stSrc.fValue;
//stDst.fValueMin := stSrc.fValueMin;
//stDst.fValueMax := stSrc.fValueMax;

F_CopyDataItemValues := TRUE;

END_FUNCTION

// ---- POUs/HMI/Utilities/DynTxt/F_CreateDynTextDefault.TcPOU
FUNCTION F_CreateDynTextDefault : ST_Text
VAR_INPUT
	wsName	: WSTRING;
END_VAR
VAR
END_VAR

F_CreateDynTextDefault.wsNameId := wsName;	
F_CreateDynTextDefault.wsName := wsName;

END_FUNCTION

// ---- POUs/System/Utilities/Functions/F_Settings_Management.TcPOU
FUNCTION F_Settings_Management : BOOL
VAR_IN_OUT
	aSettings	: ARRAY[*] OF ST_Data_Item; /// settings structure
END_VAR
VAR
	nn	: DINT;
END_VAR

//Check Array Size

FOR nn := LOWER_BOUND(aSettings, 1) TO UPPER_BOUND(aSettings, 1) DO
	IF (aSettings[nn].fValue > aSettings[nn].fValueMax) THEN
		aSettings[nn].fValue := aSettings[nn].fValueMax;
	END_IF	
	IF (aSettings[nn].fValue < aSettings[nn].fValueMin) THEN
		aSettings[nn].fValue := aSettings[nn].fValueMin;
	END_IF
	IF (aSettings[nn].nValue > aSettings[nn].fValueMax) THEN
		aSettings[nn].nValue := TO_INT(aSettings[nn].fValueMax);
	END_IF	
	IF (aSettings[nn].nValue < aSettings[nn].fValueMin) THEN
		aSettings[nn].nValue := TO_INT(aSettings[nn].fValueMin);
	END_IF	
	IF (aSettings[nn].eDataType = E_DataType.eDataType_time_ms) THEN
		IF (TO_LREAL(aSettings[nn].tValue) > aSettings[nn].fValueMax) THEN
			aSettings[nn].tValue := TO_TIME(aSettings[nn].fValueMax);
		END_IF	
		IF (TO_LREAL(aSettings[nn].tValue) < aSettings[nn].fValueMin) THEN
			aSettings[nn].tValue := TO_TIME(aSettings[nn].fValueMin);
		END_IF
	ELSIF (aSettings[nn].eDataType = E_DataType.eDataType_time_s) THEN
		IF (TO_LREAL(aSettings[nn].tValue) > (aSettings[nn].fValueMax * 1000)) THEN
			aSettings[nn].tValue := TO_TIME(aSettings[nn].fValueMax * 1000);
		END_IF	
		IF (TO_LREAL(aSettings[nn].tValue) < (aSettings[nn].fValueMin * 1000)) THEN
			aSettings[nn].tValue := TO_TIME(aSettings[nn].fValueMin * 1000);
		END_IF
	ELSIF (aSettings[nn].eDataType = E_DataType.eDataType_time_m) THEN
		IF (TO_LREAL(aSettings[nn].tValue) > (aSettings[nn].fValueMax * 60000)) THEN
			aSettings[nn].tValue := TO_TIME(aSettings[nn].fValueMax * 60000);
		END_IF	
		IF (TO_LREAL(aSettings[nn].tValue) < (aSettings[nn].fValueMin * 60000)) THEN
			aSettings[nn].tValue := TO_TIME(aSettings[nn].fValueMin * 60000);
		END_IF
	ELSIF (aSettings[nn].eDataType = E_DataType.eDataType_time_h) THEN
		IF (TO_LREAL(aSettings[nn].tValue) > (aSettings[nn].fValueMax * 360000)) THEN
			aSettings[nn].tValue := TO_TIME(aSettings[nn].fValueMax * 360000);
		END_IF	
		IF (TO_LREAL(aSettings[nn].tValue) < (aSettings[nn].fValueMin * 360000)) THEN
			aSettings[nn].tValue := TO_TIME(aSettings[nn].fValueMin * 360000);
		END_IF			
	END_IF
	IF (aSettings[nn].stName.wsNameId = "" AND aSettings[nn].stName.wsName = "") THEN
		MEMSET(ADR(aSettings[nn]), 0, SIZEOF(aSettings[nn])); // reset
	END_IF		
END_FOR

END_FUNCTION

// ---- POUs/HMI/Events/FB_EventHandler.TcPOU
FUNCTION_BLOCK FB_EventHandler IMPLEMENTS I_EventHandler
VAR_INPUT
END_VAR
VAR_OUTPUT
END_VAR
VAR
	// private instance var's
	iLog			: I_Logger;
	afbAlarm      	: ARRAY[0..Const.iMaxIdxAlam] OF FB_TcAlarm;
	fbCodeErrRef,
	fbAlarmRef      : REFERENCE TO FB_TcAlarm;
	fbMsg			: FB_TcMessage;
	fbEventLogger	: FB_TcEventLogger;
	ISb 			: I_StringBuilder;
	fbInternalSb	: FB_StringBuilder;
	iCntAlm			: INT;
	bInfoActive,
	bWarningActive,
	bErrorActive	: BOOL;
END_VAR

//ToDo: SetJsonAttribute (e.g.: error reaction)
//ToDo: F_GetEventText o.ä.
//ToDo: Listener?

// unit tests
Test();

METHOD PUBLIC ArgAddDint : I_EventHandler
VAR_INPUT
	value : DINT;
END_VAR
ArgAddDint := THIS^;
IF __ISVALIDREF(fbAlarmRef) THEN
	fbAlarmRef.ipArguments.AddDInt(value);
END_IF
END_METHOD

METHOD PUBLIC ArgAddEventRef : I_EventHandler
VAR_INPUT
	value : TcEventEntry;
END_VAR
ArgAddEventRef := THIS^;
IF __ISVALIDREF(fbAlarmRef) THEN
	fbAlarmRef.ipArguments.AddEventReferenceEx(value);
END_IF
END_METHOD

METHOD PUBLIC ArgAddLreal : I_EventHandler
VAR_INPUT
	value : LREAL;
END_VAR
ArgAddLreal := THIS^;
IF __ISVALIDREF(fbAlarmRef) THEN
	fbAlarmRef.ipArguments.AddLReal(value);
END_IF
END_METHOD

METHOD PUBLIC ArgAddString : I_EventHandler
VAR_IN_OUT CONSTANT
	value : STRING;
END_VAR
ArgAddString := THIS^;
IF __ISVALIDREF(fbAlarmRef) THEN
	fbAlarmRef.ipArguments.AddString(value);
END_IF
END_METHOD

METHOD PUBLIC ArgAddWString : I_EventHandler
VAR_IN_OUT CONSTANT
	value : WSTRING;
END_VAR
ArgAddWString := THIS^;
IF __ISVALIDREF(fbAlarmRef) THEN
	fbAlarmRef.ipArguments.AddWString(value);
END_IF
END_METHOD

METHOD PUBLIC ArgClear : I_EventHandler
ArgClear := THIS^;
IF __ISVALIDREF(fbAlarmRef) THEN
	fbAlarmRef.ipArguments.Clear();
END_IF
END_METHOD

METHOD PUBLIC ArgSbAppend : I_EventHandler
VAR_IN_OUT CONSTANT
	value : T_MaxString;
END_VAR
ArgSbAppend := THIS^;

IF ISb <> 0 THEN
	ISb.Append(value);
END_IF
END_METHOD

METHOD PUBLIC ArgSbAppendAny : I_EventHandler
VAR_INPUT
	value : ANY;
END_VAR
ArgSbAppendAny := THIS^;

IF ISb <> 0 THEN
	ISb.AppendAny(value);
END_IF
END_METHOD

METHOD PUBLIC ArgSbAppendAnyRaise : HRESULT
VAR_INPUT
	value : ANY;
END_VAR
ArgSbAppendAnyRaise := ArgSbAppendAny(value).ArgSetSbRaise();
END_METHOD

METHOD PUBLIC ArgSbAppendRaise : HRESULT
VAR_IN_OUT CONSTANT
	value : T_MaxString;
END_VAR
ArgSbAppendRaise := ArgSbAppendSet(value).Raise();
END_METHOD

METHOD PUBLIC ArgSbAppendS : I_EventHandler
VAR_INPUT
	value : T_MaxString := '';
END_VAR
ArgSbAppendS := ArgSbAppend(value);
END_METHOD

METHOD PUBLIC ArgSbAppendSet : I_EventHandler
VAR_IN_OUT CONSTANT
	value : T_MaxString;
END_VAR
ArgSbAppendSet := ArgSbAppend(value).ArgSetSb();
END_METHOD

METHOD PUBLIC ArgSbAppendWs : I_EventHandler
VAR_IN_OUT CONSTANT
	value : WSTRING;
END_VAR
ArgSbAppendWs := THIS^;

IF ISb <> 0 THEN
	ISb.AppendWs(value);
END_IF
END_METHOD

METHOD PUBLIC ArgSbAppendWsRaise : HRESULT
VAR_IN_OUT CONSTANT
	value : WSTRING;
END_VAR
ArgSbAppendWsRaise := ArgSbAppendWs(value).ArgSetSbRaise();
END_METHOD

METHOD PUBLIC ArgSbInit : I_EventHandler
VAR_IN_OUT CONSTANT
	value : T_MaxString;
END_VAR
Isb := fbInternalSb.Set(value);
ArgSbInit := THIS^;
END_METHOD

METHOD PUBLIC ArgSbInitExternal : I_EventHandler
VAR_INPUT
	sb	: I_StringBuilder;
END_VAR
ISb := sb;
ArgSbInitExternal := THIS^;
END_METHOD

METHOD PUBLIC ArgSbInitWs : I_EventHandler
VAR_IN_OUT CONSTANT
	value : WSTRING;
END_VAR
Isb := fbInternalSb.SetWs(value);
ArgSbInitWs := THIS^;
END_METHOD

METHOD PUBLIC ArgSetDint : I_EventHandler
VAR_INPUT
	value : DINT;
END_VAR
ArgSetDint := ArgClear().ArgAddDint(value);
END_METHOD

METHOD PUBLIC ArgSetEventRef : I_EventHandler
VAR_INPUT
	value : TcEventEntry;
END_VAR
ArgSetEventRef := ArgClear().ArgAddEventRef(value);
END_METHOD

METHOD PUBLIC ArgSetLreal : I_EventHandler
VAR_INPUT
	value : LREAL;
END_VAR
ArgSetLreal := ArgClear().ArgAddLreal(value);
END_METHOD

METHOD PUBLIC ArgSetSb : I_EventHandler
VAR_INPUT
	sb 		: I_StringBuilder := 0; // optional external string builder, set to 0 to use internal
END_VAR
VAR
	value	: STRING;
END_VAR
IF sb = 0 THEN
	sb := Isb;
END_IF

value := sb.ToString();
ArgSetSb := ArgClear().ArgAddString(value);
END_METHOD

METHOD PUBLIC ArgSetSbRaise : HRESULT
VAR_INPUT
	sb	: I_StringBuilder := 0; // optional external string builder, set to 0 to use internal
END_VAR
ArgSetSbRaise := ArgSetSb(sb).Raise();
END_METHOD

METHOD PUBLIC ArgSetString : I_EventHandler
VAR_IN_OUT CONSTANT
	value : STRING;
END_VAR
ArgSetString := ArgClear().ArgAddString(value);
END_METHOD

METHOD PUBLIC ArgSetWString : I_EventHandler
VAR_IN_OUT CONSTANT
	value : WSTRING;
END_VAR
ArgSetWString := ArgClear().ArgAddWString(value);
END_METHOD

METHOD PUBLIC CreateAlarm : I_EventHandler
VAR_INPUT
	stEventEntry      : TcEventEntry;
    bWithConfirmation : BOOL := FALSE;
    ipSourceInfo      : I_TcSourceInfo := NULL;
END_VAR
VAR
	hres 	: HRESULT;
	msg		: STRING;
END_VAR
CreateAlarm := THIS^;
IF (iCntAlm > Const.iMaxIdxAlam) THEN
	msg := CONCAT('Max. events exceeded, Const.iMaxIdxAlam: ', TO_STRING(Const.iMaxIdxAlam));
	fbCodeErrRef.ipArguments.Clear().AddString(msg);
	fbCodeErrRef.Raise(0);
	RETURN;
END_IF

hres := afbAlarm[iCntAlm].CreateEx(stEventEntry, bWithConfirmation, ipSourceInfo);

IF (hres = S_OK) THEN
	iCntAlm := iCntAlm + 1;
ELSE
	msg := CONCAT('Create alarm failed, HRESULT: ', TO_STRING(hres));
	fbCodeErrRef.ipArguments.Clear().AddString(msg);
	fbCodeErrRef.Raise(0);
END_IF
END_METHOD

{attribute 'monitoring' := 'call'}
PROPERTY ErrorActive : BOOL
GET
ErrorActive := bErrorActive;
END_GET
END_PROPERTY

{attribute 'monitoring' := 'call'}
PROPERTY InfoActive : BOOL
GET
InfoActive := bInfoActive;
END_GET
END_PROPERTY

METHOD Init : BOOL
iLog := SERVICES.ILog;

// init alarm event classes
CreateAlarm(TC_Events.InternalEventClass.InfoEvent);
CreateAlarm(TC_Events.InternalEventClass.WarningEvent, TRUE);
CreateAlarm(TC_Events.InternalEventClass.ErrorEvent, TRUE);
CreateAlarm(TC_Events.CodeEventClass.InfoEvent);
CreateAlarm(TC_Events.CodeEventClass.WarningEvent, TRUE);
CreateAlarm(TC_Events.CodeEventClass.ErrorEvent, TRUE);
CreateAlarm(TC_Events.SystemEventClass.InfoEvent);
CreateAlarm(TC_Events.SystemEventClass.WarningEvent, TRUE);
CreateAlarm(TC_Events.SystemEventClass.ErrorEvent, TRUE);
CreateAlarm(TC_Events.EtherCatEventClass.InfoEvent);
CreateAlarm(TC_Events.EtherCatEventClass.WarningEvent, TRUE);
CreateAlarm(TC_Events.EtherCatEventClass.ErrorEvent, TRUE);
CreateAlarm(TC_Events.EtherCatEventClass.DevicStateErrorEvent, TRUE);
CreateAlarm(TC_Events.EtherCatEventClass.LinkStateErrorEvent, TRUE);
CreateAlarm(TC_Events.HardwareEventClass.InfoEvent);
CreateAlarm(TC_Events.HardwareEventClass.WarningEvent, TRUE);
CreateAlarm(TC_Events.HardwareEventClass.ErrorEvent, TRUE);
CreateAlarm(TC_Events.TwinSafeEventClass.InfoEvent);
CreateAlarm(TC_Events.TwinSafeEventClass.WarningEvent, TRUE);
CreateAlarm(TC_Events.TwinSafeEventClass.ErrorEvent, TRUE);
CreateAlarm(TC_Events.TwinSafeEventClass.HwErrorEvent, TRUE);
CreateAlarm(TC_Events.SettingsEventClass.InfoEvent);
CreateAlarm(TC_Events.SettingsEventClass.WarningEvent, TRUE);
CreateAlarm(TC_Events.SettingsEventClass.ErrorEvent, TRUE);
CreateAlarm(TC_Events.RecipeEventClass.InfoEvent);
CreateAlarm(TC_Events.RecipeEventClass.WarningEvent, TRUE);
CreateAlarm(TC_Events.RecipeEventClass.ErrorEvent, TRUE);
CreateAlarm(TC_Events.PlantEventClass.InfoEvent);
CreateAlarm(TC_Events.PlantEventClass.WarningEvent, TRUE);
CreateAlarm(TC_Events.PlantEventClass.ErrorEvent, TRUE);

// register simple message not needed:
//CreateMessage(TC_Events.MessageEventClass.InfoEvent);

fbCodeErrRef REF= afbAlarm[0];
fbAlarmRef REF= afbAlarm[0];
END_METHOD

METHOD PUBLIC Raise : HRESULT
VAR_INPUT
	nTimeStamp : ULINT := 0;
END_VAR
IF NOT __ISVALIDREF(fbAlarmref) THEN 
	Raise := S_FALSE;
	RETURN;	
END_IF

bInfoActive := fbAlarmRef.eSeverity >= TcEventSeverity.Info;
bWarningActive := fbAlarmRef.eSeverity >= TcEventSeverity.Warning;
bErrorActive := fbAlarmRef.eSeverity >= TcEventSeverity.Error;
Raise := fbAlarmref.Raise(nTimeStamp);
END_METHOD

METHOD PUBLIC Reset : BOOL
VAR_INPUT
END_VAR
fbEventLogger.ConfirmAllAlarms();
fbEventLogger.ClearAllAlarms();
fbEventLogger.ClearLoggedEvents(0);

bInfoActive :=
bWarningActive :=
bErrorActive := FALSE;
END_METHOD

METHOD PUBLIC Select : I_EventHandler
VAR_INPUT
	stEventEntry : TcEventEntry;
END_VAR
VAR
	hres : HRESULT;
END_VAR
Select := THIS^;
fbAlarmRef REF= afbAlarm[0];
hres := fbEventLogger.GetAlarmEx(stEventEntry, 0, fbAlarmRef);
IF hres <> S_OK OR NOT __ISVALIDREF(fbAlarmRef) THEN
	fbAlarmRef REF= afbAlarm[0];
END_IF
END_METHOD

METHOD PUBLIC Send : BOOL
VAR_INPUT
	stEventEntry      : TcEventEntry;
    ipSourceInfo      : I_TcSourceInfo := NULL;
    nTimeStamp        : ULINT := 0;
    ipArguments       : I_TcArguments := NULL;
END_VAR
Send := fbEventLogger.SendMessageEx(stEventEntry, ipSourceInfo, nTimeStamp, ipArguments) = S_OK;
END_METHOD

METHOD PUBLIC SendJson : BOOL
VAR_INPUT
	stEventEntry      : TcEventEntry;
    ipSourceInfo      : I_TcSourceInfo := NULL;
    nTimeStamp        : ULINT := 0;
    ipArguments       : I_TcArguments := NULL;
END_VAR
VAR_IN_OUT CONSTANT
    sJsonAttribute    : STRING;
END_VAR
SendJson := fbEventLogger.SendMessageEx2(stEventEntry, ipSourceInfo, nTimeStamp, ipArguments, sJsonAttribute) = S_OK;
END_METHOD

METHOD PUBLIC SendString : BOOL
VAR_IN_OUT CONSTANT
	msg : STRING;	
END_VAR
VAR_INST
	args : FB_TcArguments;
END_VAR
SendString := Send(TC_EVENTS.MessageEventClass.InfoEvent, NULL, 0, 
													args.Clear().AddString(msg));
END_METHOD

METHOD PUBLIC SendStringJson : BOOL
VAR_IN_OUT CONSTANT
	msg				: STRING;
	sJsonAttribute	: STRING;
END_VAR
VAR_INST
	args 			: FB_TcArguments;
END_VAR
SendStringJson := SendJson(TC_EVENTS.MessageEventClass.InfoEvent, NULL, 0, 
													args.Clear().AddString(msg), 
													sJsonAttribute);
END_METHOD

METHOD PRIVATE Test : BOOL
VAR_INST
	// event alarm test
	iTestCase		: INT;
	bAlarmTest, 
	bMsgTest,
	bClearAlarmTest : BOOL;
	HRES			: HRESULT;
END_VAR
// alarm tests
IF bAlarmTest THEN
	bAlarmTest := FALSE;
	IF iTestCase = 0 THEN
		HRES := fbEventLogger.GetAlarmEx(TC_Events.CodeEventClass.ErrorEvent, 0, fbAlarmRef);
		IF (HRES <> 0 OR  NOT __ISVALIDREF(fbAlarmRef)) THEN RETURN; END_IF
		iTestCase := 10;
		fbAlarmRef.ipArguments.Clear().AddString('check bounds');
		fbAlarmRef.Raise(0);
		
	ELSIF iTestCase = 1 THEN
		Select(TC_Events.CodeEventClass.ErrorEvent)
			  .ArgSetString('check bounds')
			  .Raise();
		RETURN;
	ELSIF iTestCase = 2 THEN
		Select(TC_Events.HardwareEventClass.ErrorEvent)
			  .ArgSetString('div 0')
			  .Raise();
	ELSIF iTestCase = 3 THEN		
		Select(TC_Events.HardwareEventClass.WarningEvent)
			  .ArgSetString('check pointer')
			  .Raise();
	ELSIF iTestCase = 4 THEN
		// adding localizable argument sample 
		Select(TC_Events.SettingsEventClass.InfoEvent)
			  .ArgSetEventRef(TC_Events.TranslationListEventClass.TranslationListEventClass_NameEvent)
			  .ArgAddString('sdc')
			  .Raise();
	END_IF
	
	//fbAlarm.eConfirmationState = TcEventConfirmationState.WaitForConfirmation
	//fbAlarm.bActive
END_IF

// simple message tests
IF bMsgTest THEN
	bMsgTest := FALSE;
	IF iTestCase = 0 THEN
		SendString('Rezept wurde geladen!');
	ELSIF iTestCase = 2 THEN
		SendString('Rezept wurde gespeichert!');
	ELSIF iTestCase = 3 THEN
		SendString('Rezept wurde kopiert!');
	ELSE
		Send(TC_Events.MessageEventClass.InfoEvent, Null, 0, fbMsg.ipArguments);
	END_IF
	
	//fbMsg.Send();
END_IF

// reset/clear alarms
IF bClearAlarmTest THEN
	bClearAlarmTest := FALSE;
	Reset();
END_IF
END_METHOD

{attribute 'monitoring' := 'call'}
PROPERTY WarningActive : BOOL
GET
WarningActive := bWarningActive;
END_GET
END_PROPERTY

END_FUNCTION_BLOCK

// ---- POUs/System/Utilities/String/FB_StringBuilder.TcPOU
FUNCTION_BLOCK FB_StringBuilder IMPLEMENTS I_StringBuilder
VAR_INPUT
END_VAR
VAR_OUTPUT
END_VAR
VAR
    sString : T_MaxString;
END_VAR

///
/// String Builder Fluent-Code Style
/// Credits to Gerhard Barteling, https://www.plccoder.com/fluent-code/
///

METHOD PUBLIC Append : I_StringBuilder // Append text to the current build string.
VAR_IN_OUT CONSTANT
	text : T_MaxString; // Text to append to current build string
END_VAR
sString := Concat(sString, text);
Append := THIS^;
END_METHOD

METHOD PUBLIC AppendAny : I_StringBuilder // Append text to the current build string.
VAR_INPUT
	value : ANY; // Value to append to current build string
END_VAR
VAR
	pSTR	: POINTER TO STRING;
	pWSTR	: POINTER TO WSTRING;
	pBOOL	: POINTER TO BOOL;
	pBYTE	: POINTER TO BYTE;
	pWORD	: POINTER TO WORD;
	pDWORD	: POINTER TO DWORD;
	pLWORD	: POINTER TO LWORD;
	pSINT	: POINTER TO SINT;
	pINT	: POINTER TO INT;
	pDINT	: POINTER TO DINT;
	pLINT	: POINTER TO LINT;
	pUSINT	: POINTER TO USINT;
	pUINT	: POINTER TO UINT;
	pUDINT	: POINTER TO UDINT;
	pULINT	: POINTER TO ULINT;
	pREAL	: POINTER TO REAL;
	pLREAL	: POINTER TO LREAL;
	pTIME	: POINTER TO TIME;
	pLTIME	: POINTER TO LTIME;
	pDATE	: POINTER TO DATE;
	pDT		: POINTER TO DT;
	pTOD	: POINTER TO TOD;
	pENUM	: POINTER TO ENUM;
END_VAR
CASE value.TypeClass OF
	__SYSTEM.TYPE_CLASS.TYPE_STRING: 
		pSTR := value.pValue;
		sString:= CONCAT(sString, TO_STRING(pSTR^));
		
	__SYSTEM.TYPE_CLASS.TYPE_WSTRING:
		pWSTR := value.pValue;
		sString:= CONCAT(sString, TO_STRING(pWSTR^));
		
	__SYSTEM.TYPE_CLASS.TYPE_BOOL:
		pBOOL := value.pValue;
		sString:= CONCAT(sString, TO_STRING(pBOOL^));
		
	__SYSTEM.TYPE_CLASS.TYPE_BYTE:
		pBYTE := value.pValue;
		sString:= CONCAT(sString, TO_STRING(pBYTE^));
		
	__SYSTEM.TYPE_CLASS.TYPE_WORD:
		pWORD := value.pValue;
		sString:= CONCAT(sString, TO_STRING(pWORD^));
		
	__SYSTEM.TYPE_CLASS.TYPE_DWORD:
		pDWORD := value.pValue;
		sString:= CONCAT(sString, TO_STRING(pDWORD^));
		
	__SYSTEM.TYPE_CLASS.TYPE_LWORD:
		pLWORD := value.pValue;
		sString:= CONCAT(sString, TO_STRING(pLWORD^));
		
	__SYSTEM.TYPE_CLASS.TYPE_SINT:
		pSINT := value.pValue;
		sString:= CONCAT(sString, TO_STRING(pSINT^));
		
	__SYSTEM.TYPE_CLASS.TYPE_INT:
		pINT := value.pValue;
		sString:= CONCAT(sString, TO_STRING(pINT^));
		
	__SYSTEM.TYPE_CLASS.TYPE_DINT:
		pDINT := value.pValue;
		sString:= CONCAT(sString, TO_STRING(pDINT^));
		
	__SYSTEM.TYPE_CLASS.TYPE_LINT:
		pLINT := value.pValue;
		sString:= CONCAT(sString, TO_STRING(pLINT^));
		
	__SYSTEM.TYPE_CLASS.TYPE_USINT:
		pUSINT := value.pValue;
		sString:= CONCAT(sString, TO_STRING(pUSINT^));
		
	__SYSTEM.TYPE_CLASS.TYPE_UINT:
		pUINT := value.pValue;
		sString:= CONCAT(sString, TO_STRING(pUINT^));
		
	__SYSTEM.TYPE_CLASS.TYPE_UDINT:
		pUDINT := value.pValue;
		sString:= CONCAT(sString, TO_STRING(pUDINT^));
		
	__SYSTEM.TYPE_CLASS.TYPE_ULINT:
		pULINT := value.pValue;
		sString:= CONCAT(sString, TO_STRING(pULINT^));
		
	__SYSTEM.TYPE_CLASS.TYPE_REAL:
		pREAL := value.pValue;
		sString:= CONCAT(sString, TO_STRING(pREAL^));
		
	__SYSTEM.TYPE_CLASS.TYPE_LREAL:
		pLREAL := value.pValue;
		sString:= CONCAT(sString, TO_STRING(pLREAL^));
		
	__SYSTEM.TYPE_CLASS.TYPE_TIME:
		pTIME := value.pValue;
		sString:= CONCAT(sString, TO_STRING(pTIME^));
		
	__SYSTEM.TYPE_CLASS.TYPE_LTIME:
		pLTIME := value.pValue;
		sString:= CONCAT(sString, TO_STRING(pLTIME^));
	
	__SYSTEM.TYPE_CLASS.TYPE_DATE:
		pDATE := value.pValue;
		sString:= CONCAT(sString, TO_STRING(pDATE^));
		
	__SYSTEM.TYPE_CLASS.TYPE_DATEANDTIME:
		pDT := value.pValue;
		sString:= CONCAT(sString, TO_STRING(pDT^));
		
	__SYSTEM.TYPE_CLASS.TYPE_TIMEOFDAY:
		pTOD := value.pValue;
		sString:= CONCAT(sString, TO_STRING(pTOD^));
		
	__SYSTEM.TYPE_CLASS.TYPE_ENUM: // does not work!
		pENUM := value.pValue;
		sString:= CONCAT(sString, TO_STRING(pENUM^));

END_CASE

AppendAny := THIS^;
END_METHOD

METHOD PUBLIC AppendWs : I_StringBuilder
VAR_IN_OUT CONSTANT
	value : WSTRING;
END_VAR
VAR
	str	  : STRING;
END_VAR
WSTRING_TO_STRING2(ADR(str), ADR(value), SIZEOF(str));
sString := Concat(sString, str);
AppendWs := THIS^;
END_METHOD

METHOD PUBLIC Clear : I_StringBuilder // Clear the current build string.
VAR_INPUT
END_VAR
sString := '';
Clear := THIS^;
END_METHOD

METHOD PUBLIC Insert : I_StringBuilder
VAR_INPUT
	text	 : T_MaxString;	// Text to append to current build string
	position : INT;			// Insert position (Index)
END_VAR
sString := Tc2_Standard.INSERT(sString, text, position);
Insert := THIS^;
END_METHOD

METHOD PUBLIC Reset : I_StringBuilder //Reset current build string to an empty string.
VAR_INPUT
END_VAR
sString := '';
Reset := THIS^;
END_METHOD

METHOD PUBLIC Set : I_StringBuilder
VAR_INPUT
	text : T_MaxString; //Text to append to current build string
END_VAR
sString := text;
Set := THIS^;
END_METHOD

METHOD PUBLIC SetWs : I_StringBuilder
VAR_IN_OUT CONSTANT
	value : WSTRING;
END_VAR
SetWs := Clear().AppendWs(value);
END_METHOD

METHOD PUBLIC ToString : T_MaxString // Returns current build string.
VAR_INPUT
END_VAR
ToString := sString;
END_METHOD

END_FUNCTION_BLOCK

// ---- POUs/System/Supervision/P_Supervision.TcPOU
/// Supervision function block - system watchdog
PROGRAM INTERNAL P_Supervision
VAR_IN_OUT
	/// Safets IOs
	stIO_Cabinet		: ST_ControlCabinetIO;
		
	/// Logger
	nLogger				: I_Logger;
END_VAR
VAR_INPUT
END_VAR
VAR_OUTPUT
	bError				: BOOL;	
	bWarning			: BOOL;
	
	bCycleStop			: BOOL;
	bFastStop			: BOOL;
END_VAR
VAR
	/// event handler
	IEvent			: I_EventHandler;
	
	/// Hardware diag FB
	fbDiagEtherCAT	: FB_DiagEtherCAT;
	
	/// private var's
	aa									: INT;	
	rTrigMachineStop_Cycle				: R_TRIG;
	rTrigMachineStop_Fast				: R_TRIG;
	tonRstStillstw						: TON;
END_VAR

/// 
/// supervision function block of the project
/// 

// reset

// run supervision (ES, Safety signals, IO-errors, etc.)

// HW diagnostics
M_EcSupervision();
M_ControlCabinet_A01();

// task cycle time exceeded
IF Statics.stPlcSystemInfo.stPlcTaskSystemInfo.CycleTimeExceeded THEN
	IEvent.Select(TC_Events.SystemEventClass.ErrorEvent)
		  .ArgSetWString(stTextListGlobal.stText_System.stText_CycletimeExceeded.wsName)
		  .Raise();	
END_IF


//-------------------------------------------------------------------------------------------------------------

IF HMI.stHmi.stIn.stMain.stButton_Start.bClick AND NOT stGlobalModuleInfo.bStation_All_Auto AND P_Safety.OpMode_Auto THEN
	IEvent.Select(TC_Events.SystemEventClass.InfoEvent)
		  .ArgSetString('Start Auto nicht moeglich -> Station nicht in Betriebsart Auto')
		  .Raise();
END_IF


//-------------------------------------------------------------------------------------------------------------

IF HMI.stHmi.stIn.stMain.stButton_Start.bClick AND NOT P_Safety.OpMode_Auto THEN
	IEvent.Select(TC_Events.SystemEventClass.InfoEvent)
		  .ArgSetString('Start Auto nicht moeglich -> Schlüsselschalter nicht auf Auto')
		  .Raise();
END_IF


//ToDo: stop / fast stop on alarm trigger
//rTrigMachineStop_Cycle(CLK := Services.fbNotiHandler.stNotificationData.eAlarmStopMode = E_EventReaction.CycleStop, Q => bCycleStop);
//rTrigMachineStop_Fast(CLK := Services.fbNotiHandler.stNotificationData.eAlarmStopMode = E_EventReaction.Stop, Q => bFastStop);

/// System error level
{attribute 'monitoring' := 'call'}
PROPERTY Error : BOOL
GET // INTERNAL
Error := bError;
END_GET
END_PROPERTY

METHOD PRIVATE M_ControlCabinet_A01 : BOOL
VAR_INPUT
END_VAR
// EC-Error
IF IO.stControlCabinetIO.stIn.IarrEcStates[E_EtherCatBox.eEtherCatBox_ControlCabinet] <> 8 THEN
	IEvent.Select(TC_Events.EtherCatEventClass.ErrorEvent)
		  .ArgSetString('EtherCatBox Control Cabinet | EC State Error')
		  .Raise();
ELSIF IO.stControlCabinetIO.stIn.IarrEcStates[E_EtherCatBox.eEtherCatBox_Oven_A] <> 8 THEN
	IEvent.Select(TC_Events.EtherCatEventClass.ErrorEvent)
		  .ArgSetString('EtherCatBox Oven A | EC State Error')
		  .Raise();
ELSIF IO.stControlCabinetIO.stIn.IarrEcStates[E_EtherCatBox.eEtherCatBox_Oven_B] <> 8 THEN
	IEvent.Select(TC_Events.EtherCatEventClass.ErrorEvent)
		  .ArgSetString('EtherCatBox Oven B | EC State Error')
		  .Raise();
ELSIF IO.stControlCabinetIO.stIn.IarrEcStates[E_EtherCatBox.eEtherCatBox_Storage] <> 8 THEN
	IEvent.Select(TC_Events.EtherCatEventClass.ErrorEvent)
		  .ArgSetString('EtherCatBox Storage | EC State Error')
		  .Raise();
END_IF
			  
(*	24V-Versorgung Netzgerät 1 Schutzschalter	
ELSIF NOT IO.stControlCabinetIO.stIn.stA01.b24V_NetzSchutz1Ok THEN
	IEvent.Select(TC_Events.HardwareEventClass.ErrorEvent)
			  .ArgSetString('=A01.G10-1QA1 | 24V-Versorgung Netzgerät 1 Schutzschalter NOK')
			  .Raise();
END_IF
*)
END_METHOD

METHOD PRIVATE M_EcSupervision : BOOL
VAR_INPUT
END_VAR
VAR_INST

END_VAR

// automatic EC supervision
fbDiagEtherCAT();

(*
//IarrEcState
// Diag EC Boxes for fast reaction				
IF (stIO_Cabinet.stIn.IarrEcStates[1] <> 8) THEN
	bError:=TRUE;
	fbNotiHandler.M_SetNotificationEx(F_CreateDynText("403",403),
									stTextListGlobal.stText_NG_Hardware, 
									stTextListGlobal.stText_EtherCatBox_Error, "++M1+E2-57CO1 (CU1128)", stTextListGlobal.stText_EtherCatBox_OP_Error, 
									E_AlarmPriority.Error, E_NotificationMode.eNotificationMode_Reset);	
END_IF
IF (stIO_Cabinet.stIn.IarrEcStates[2] <> 8) THEN
	bError:=TRUE;
	fbNotiHandler.M_SetNotificationEx(F_CreateDynText("404",404),
									stTextListGlobal.stText_NG_Hardware, 
									stTextListGlobal.stText_EtherCatBox_Error, "++M1+E2-57CO1 (CU1128-B)", stTextListGlobal.stText_EtherCatBox_OP_Error, 
									E_AlarmPriority.Error, E_NotificationMode.eNotificationMode_Reset);	
END_IF
IF (stIO_Cabinet.stIn.IarrEcStates[3] <> 8) THEN
	bError:=TRUE;
	fbNotiHandler.M_SetNotificationEx(F_CreateDynText("405",405),
									stTextListGlobal.stText_NG_Hardware, 
									stTextListGlobal.stText_EtherCatBox_Error, "++M1+E2-57CO1 (CU1128-C)", stTextListGlobal.stText_EtherCatBox_OP_Error, 
									E_AlarmPriority.Error, E_NotificationMode.eNotificationMode_Reset);	
END_IF
IF (stIO_Cabinet.stIn.IarrEcStates[4] <> 8) THEN
	bError:=TRUE;
	fbNotiHandler.M_SetNotificationEx(F_CreateDynText("406",406),
									stTextListGlobal.stText_NG_Hardware, 
									stTextListGlobal.stText_EtherCatBox_Error, "++M1+E2-62BC1 (EK1100)", stTextListGlobal.stText_EtherCatBox_OP_Error, 
									E_AlarmPriority.Error, E_NotificationMode.eNotificationMode_Reset);	
END_IF
IF (stIO_Cabinet.stIn.IarrEcStates[5] <> 8) THEN
	bError:=TRUE;
	fbNotiHandler.M_SetNotificationEx(F_CreateDynText("407",407),
									stTextListGlobal.stText_NG_Hardware, 
									stTextListGlobal.stText_EtherCatBox_Error, "++A1+P1-4A2 (EP2338-0002)", stTextListGlobal.stText_EtherCatBox_OP_Error, 
									E_AlarmPriority.Error, E_NotificationMode.eNotificationMode_Reset);	
END_IF
IF (stIO_Cabinet.stIn.IarrEcStates[6] <> 8) THEN
	bError:=TRUE;
	fbNotiHandler.M_SetNotificationEx(F_CreateDynText("0",0),
									stTextListGlobal.stText_NG_Hardware, 
									stTextListGlobal.stText_EtherCatBox_Error, "++A1+P1-5SI0 (EP1908)", stTextListGlobal.stText_EtherCatBox_OP_Error, 
									E_AlarmPriority.Error, E_NotificationMode.eNotificationMode_Reset);	
END_IF
IF (stIO_Cabinet.stIn.IarrEcStates[7] <> 8)  THEN
	bError:=TRUE;
	fbNotiHandler.M_SetNotificationEx(F_CreateDynText("408",408),
									stTextListGlobal.stText_NG_Hardware, 
									stTextListGlobal.stText_EtherCatBox_Error, "++A1+P1-6SI0 (EP1908)", stTextListGlobal.stText_EtherCatBox_OP_Error, 
									E_AlarmPriority.Error, E_NotificationMode.eNotificationMode_Reset);	
END_IF
IF (stIO_Cabinet.stIn.IarrEcStates[8] <> 8) THEN
	bError:=TRUE;
	fbNotiHandler.M_SetNotificationEx(F_CreateDynText("409",409),
									stTextListGlobal.stText_NG_Hardware, 
									stTextListGlobal.stText_EtherCatBox_Error, "++A1+P1-3A2 (EP2338-0002)", stTextListGlobal.stText_EtherCatBox_OP_Error, 
									E_AlarmPriority.Error, E_NotificationMode.eNotificationMode_Reset);	
END_IF

IF (stIO_Cabinet.stIn.IarrEcStates[9] <> 8) THEN
	bError:=TRUE;
	fbNotiHandler.M_SetNotificationEx(F_CreateDynText("410",410),
									stTextListGlobal.stText_NG_Hardware, 
									stTextListGlobal.stText_EtherCatBox_Error, "++M1+E1-46BC3 (EK1100)", stTextListGlobal.stText_EtherCatBox_OP_Error, 
									E_AlarmPriority.Error, E_NotificationMode.eNotificationMode_Reset);	
END_IF
IF (stIO_Cabinet.stIn.IarrEcStates[10] <> 8) THEN
	bError:=TRUE;
	fbNotiHandler.M_SetNotificationEx(F_CreateDynText("411",411),
									stTextListGlobal.stText_NG_Hardware, 
									stTextListGlobal.stText_EtherCatBox_Error, "++M1+E1-38U1 (AX5206-0000-0213)", stTextListGlobal.stText_EtherCatBox_OP_Error, 
									E_AlarmPriority.Error, E_NotificationMode.eNotificationMode_Reset);	
END_IF
IF (stIO_Cabinet.stIn.IarrEcStates[11] <> 8) THEN
	bError:=TRUE;
	fbNotiHandler.M_SetNotificationEx(F_CreateDynText("412",412),
									stTextListGlobal.stText_NG_Hardware, 
									stTextListGlobal.stText_EtherCatBox_Error, "++M1+E1-31U1 (Rtt)", stTextListGlobal.stText_EtherCatBox_OP_Error, 
									E_AlarmPriority.Error, E_NotificationMode.eNotificationMode_Reset);	
END_IF
IF (stIO_Cabinet.stIn.IarrEcStates[12] <> 8) THEN
	bError:=TRUE;
	fbNotiHandler.M_SetNotificationEx(F_CreateDynText("413",413),
									stTextListGlobal.stText_NG_Hardware, 
									stTextListGlobal.stText_EtherCatBox_Error, "++M1+Festo_V1 (CPX-FB37)", stTextListGlobal.stText_EtherCatBox_OP_Error, 
									E_AlarmPriority.Error, E_NotificationMode.eNotificationMode_Reset);	
END_IF
IF (stIO_Cabinet.stIn.IarrEcStates[13] <> 8) THEN
	bError:=TRUE;
	fbNotiHandler.M_SetNotificationEx(F_CreateDynText("414",414),
									stTextListGlobal.stText_NG_Hardware, 
									stTextListGlobal.stText_EtherCatBox_Error, "++M1+KeyenceSR_X100-30U1 (SR-EC1)", stTextListGlobal.stText_EtherCatBox_OP_Error, 
									E_AlarmPriority.Error, E_NotificationMode.eNotificationMode_Reset);	
END_IF
*)
END_METHOD

METHOD INTERNAL M_Init : BOOL
VAR_INPUT
END_VAR
SetReferences(Services.fbEventHandler);
END_METHOD

/// resets all notification flags and reset-needed state 
METHOD M_Reset
VAR
	ii: INT;
END_VAR
// reset error level
nLogger.AddLog(Concat2x('Reset, Error: ', TO_STRING(bError)), 'Supervision', eLogLevel_info);
bError := FALSE;
bWarning := FALSE;
END_METHOD

/// Dependency injection method.
{attribute 'object_name' := 'SetReferences'}
METHOD INTERNAL SetReferences
VAR_INPUT
	/// event access provider
	IEventHandler : I_EventHandler;
END_VAR
// init components stuff here...
IEvent := IEventHandler;
fbDiagEtherCAT.SetReferences(IEvent);
END_METHOD

END_PROGRAM

// ---- POUs/System/Supervision/EtherCAT/FB_DiagEtherCAT.TcPOU
FUNCTION_BLOCK FB_DiagEtherCAT
VAR_OUTPUT
	/// EtherCAT bus state ok
	bBusStatus_EtherCatOk	: BOOL := TRUE;
	stTextDeviceState		: ST_Text;
	stTextLinkState			: ST_Text;
	stTextBmk				: ST_Text;
END_VAR
VAR
	/// EtherCAT Master inputs
	aEcMasters AT%I*		: ARRAY[0..Const.iMaxIdxEcMaster] OF ST_EcMaster_In;
	
	/// event handler reference
	IEvent : I_EventHandler;
	
	// EtherCat bus with an error
	nSelectedMaster				: INT;
	// Slave number with an error
	nError_EcSlaveNr			: INT;
	//AmsNetId of the EtherCAT master device
	sEcMasterNetId				: T_AmsNetId;
	// Get all slave address
	fbEcGetAllSlaveAddr			: FB_EcGetAllSlaveAddr;
	// Get all slave states
	fbEcGetAllSlaveStates		: FB_EcGetAllSlaveStates;

	// Get slave name
	fbGetSlaveName 				: IOF_GetBoxNameByAddr;
	
	arrSlaves					: ARRAY[0..iMaxIdxDiagSlave] OF UINT;
	arrSlaveState				: ARRAY[0..iMaxIdxDiagSlave] OF ST_EcSlaveState;
	nIdx						: INT;
	
	nStep				: INT;
	tonCycle			: TON;
	tonDelay_NewCycle	: TON;
	nSearchErrCount		: INT;
	ii					: INT;
	
	bErrorFound			: BOOL;
	sb					: FB_StringBuilder;
END_VAR
VAR CONSTANT
	iMaxIdxDiagSlave	: INT := 2000;
END_VAR

// chk reference
IF iEvent = 0 THEN
	RETURN;
END_IF

// chk EtherCAT master linked (device state, device ID, Ams addres)
IF NOT M_CheckEcHwLinked() THEN
	RETURN;
END_IF

// call timer
tonCycle(PT := T#1S);
tonCycle.IN := FALSE;

tonDelay_NewCycle(PT := T#10S);
tonDelay_NewCycle.IN := FALSE;

// chk EtherCAT bus error
IF nStep = 0 AND bBusStatus_EtherCatOk THEN
	FOR ii := 0 TO Const.iMaxIdxEcMaster DO
		IF aEcMasters[ii].nDeviceState <> 0 THEN
			nSelectedMaster := ii;
			bBusStatus_EtherCatOk := FALSE;
			stTextDeviceState := M_ConvertEcMasterStateToText(aEcMasters[ii].nDeviceState);
			IEvent.Select(TC_Events.EtherCatEventClass.ErrorEvent)
		  		  .ArgSetSbRaise(sb.SetWs(stTextDeviceState.wsName).Append('Master ID: ').AppendAny(aEcMasters[ii].nDevId));
			EXIT;
		END_IF
	END_FOR
END_IF

// select master
nSelectedMaster := LIMIT(0, nSelectedMaster, Const.iMaxIdxEcMaster);

// get masters NetId
sEcMasterNetId := F_CreateAmsNetId(nIds := aEcMasters[nSelectedMaster].stAmsAdr.netId);

// Diagnose the bus participants
CASE nStep OF
	0:
		// wait cycle
		tonCycle.IN := TRUE;
		IF tonCycle.Q THEN
			// no error
			//IF refMasIn.stSystem.aEcMasters[nSelectedMaster].nDeviceState = 0 THEN
				//bBusStatus_EtherCatOk := TRUE;
			// reset diagnose
			//ELSIF NOT bBusStatus_EtherCatOk THEN
				fbEcGetAllSlaveAddr(sNetId:= sEcMasterNetId ,
									pAddrBuf:= ADR(arrSlaves),
									cbBufLen:= SIZEOF(arrSlaves),
									bExecute:= FALSE );
				nError_EcSlaveNr := 0;//-1;
				nIdx := 0;
				nSearchErrCount := 0;
				nStep := 20;
			//END_IF
		END_IF

	20:
		// read out slave addresses
		fbEcGetAllSlaveAddr(sNetId:= sEcMasterNetId ,
							pAddrBuf:= ADR(arrSlaves),
							cbBufLen:= SIZEOF(arrSlaves),
							bExecute:= TRUE );
		IF fbEcGetAllSlaveAddr.bBusy THEN
			nStep := 30;
		ELSIF fbEcGetAllSlaveAddr.bError THEN
			nStep := 1000;
		END_IF

	30:
		// wait until reading is finished
		fbEcGetAllSlaveAddr(sNetId:= sEcMasterNetId ,
							pAddrBuf:= ADR(arrSlaves),
							cbBufLen:= SIZEOF(arrSlaves),
							bExecute:= TRUE );
		IF NOT fbEcGetAllSlaveAddr.bBusy AND NOT fbEcGetAllSlaveAddr.bError THEN
			fbEcGetAllSlaveAddr(sNetId:= sEcMasterNetId ,
								pAddrBuf:= ADR(arrSlaves),
								cbBufLen:= SIZEOF(arrSlaves),
								bExecute:= FALSE );
			nStep := 100;
		ELSIF fbEcGetAllSlaveAddr.bError THEN
			nStep := 1000;
		END_IF

(*	Get all slave states	*) 
	100:
		fbEcGetAllSlaveStates(	sNetId:= sEcMasterNetId,
								pStateBuf := ADR(arrSlaveState),
								cbBufLen  := SIZEOF(arrSlaveState),
								bExecute:= FALSE );
		IF NOT fbEcGetAllSlaveStates.bBusy THEN
			nIdx := 0;
			nStep := 110;
		END_IF

	110:
		// read out slave states
		fbEcGetAllSlaveStates(	sNetId:= sEcMasterNetId,
								pStateBuf := ADR(arrSlaveState),
								cbBufLen  := SIZEOF(arrSlaveState),
								bExecute:= TRUE );
		IF fbEcGetAllSlaveStates.bBusy THEN
			nStep := 120;
		ELSIF fbEcGetAllSlaveStates.bError THEN
			nStep := 1000;
		END_IF
		
	120:
		// wait until reading is finished
		fbEcGetAllSlaveStates(	sNetId:= sEcMasterNetId,
								pStateBuf := ADR(arrSlaveState),
								cbBufLen  := SIZEOF(arrSlaveState),
								bExecute:= TRUE );
		IF NOT fbEcGetAllSlaveStates.bBusy AND NOT fbEcGetAllSlaveStates.bError THEN
			fbEcGetAllSlaveStates(	sNetId:= sEcMasterNetId,
									pStateBuf := ADR(arrSlaveState),
									cbBufLen  := SIZEOF(arrSlaveState),
									bExecute:= FALSE );
			nStep := 200;
		ELSIF fbEcGetAllSlaveStates.bError THEN
			nStep := 1000;
		END_IF
		
(*	Evaluate	*)
	200:
		// search slaves for faulty status
		bErrorFound := FALSE;
		FOR ii := 0 TO iMaxIdxDiagSlave DO
			IF arrSlaves[ii] = 0 THEN
				EXIT;
			ELSIF arrSlaveState[ii].deviceState <> EC_DEVICE_STATE_OP OR arrSlaveState[ii].linkState <> EC_LINK_STATE_OK THEN
				nError_EcSlaveNr := ii;
				stTextDeviceState := M_ConvertEcDeviceStateToText(arrSlaveState[ii].deviceState);
				stTextLinkState := M_ConvertEcLinkStateToText(arrSlaveState[ii].linkState);
				bErrorFound := TRUE;
				EXIT;
			END_IF
		END_FOR
		
		// Error found -> read out boxname
		IF bErrorFound THEN
			bBusStatus_EtherCatOk := FALSE;
			nStep := 300;
		ELSE
			bBusStatus_EtherCatOk := TRUE;
			nStep := 0;
		END_IF
		
		
		(*
		// Error found -> read out boxname
		IF bErrorFound THEN
			bBusStatus_EtherCatOk := FALSE;
			nStep := 300;
		// Error not found after repeated searches -> wait a while
		ELSIF nSearchErrCount > 3 THEN
			nStep := 1000;
		// read out the status again
		ELSE
			nSearchErrCount := nSearchErrCount + 1;
			nStep := 100;
		END_IF
		*)
		
	
(*	Detail Diagnose	*)
	300:
		fbGetSlaveName(	NETID		:= '',	(*local*)
						DEVICEID	:= aEcMasters[nSelectedMaster].nDevId,
						BOXADDR		:= arrSlaves[nError_EcSlaveNr],
						START		:= FALSE);
		IF NOT fbGetSlaveName.Busy THEN
			nStep := 310;
		END_IF

	310:
		// read out term
		fbGetSlaveName(NETID		:= '',	(*local*)
						DEVICEID	:= aEcMasters[nSelectedMaster].nDevId,
						BOXADDR		:= arrSlaves[nError_EcSlaveNr],          
						START		:= TRUE);
		IF fbGetSlaveName.Busy AND NOT fbGetSlaveName.ERR THEN
			nStep := 320;
		ELSIF fbGetSlaveName.ERR THEN
			nStep := 1000;
		END_IF

	320:
		// wait until reading is finished
		fbGetSlaveName(NETID		:= '',	(*local*)
						DEVICEID	:= aEcMasters[nSelectedMaster].nDevId,
						BOXADDR		:= arrSlaves[nError_EcSlaveNr],
						START		:= TRUE);
		IF NOT fbGetSlaveName.Busy AND NOT fbGetSlaveName.ERR THEN
			stTextBmk := F_CreateDynTextDefault(WCONCAT("BMK: ", STRING_TO_WSTRING(fbGetSlaveName.BOXNAME)));
			fbGetSlaveName(	NETID		:= '',	(*local*)
							DEVICEID	:= aEcMasters[nSelectedMaster].nDevId,
							BOXADDR		:= arrSlaves[nError_EcSlaveNr],
							START		:= FALSE);
			nStep := 350;
		ELSIF fbGetSlaveName.ERR THEN
			nStep := 1000;
		END_IF

(*	Create and output error text	*)
	350:
		
		IEvent.Select(TC_Events.EtherCatEventClass.ErrorEvent)
		  	  .ArgSetSbRaise(sb.SetWs(stTextListGlobal.stText_System.stText_EC_CommonError.wsName).AppendWs(stTextBmk.wsName));
//		IEvent.Select(TC_Events.EcDevicStateError, E_Priority.ePriority_fault, stTextDeviceState, stTextBmk).Raise();
//		IEvent.Select(TC_Events.EcLinkStateError, E_Priority.ePriority_fault, stTextLinkState, stTextBmk).Raise();

		// wait a few seconds before next search
		nStep := 1000;


(*	ERROR	*)
	1000:
		// new trial
		tonDelay_NewCycle.IN := TRUE;
		IF tonDelay_NewCycle.Q THEN
			nStep := 0;
		END_IF

END_CASE

METHOD PRIVATE M_CheckEcHwLinked : BOOL
VAR_INST
	bChkEcHwLinked : BOOL;
END_VAR
IF bChkEcHwLinked THEN
	M_CheckEcHwLinked := TRUE;
	RETURN;
END_IF

// chk EtherCAT master linked (device state, device ID, Ams addres)
bChkEcHwLinked := TRUE;
FOR ii := 0 TO Const.iMaxIdxEcMaster DO
	IF aEcMasters[ii].nDevId = 0 THEN
		IEvent.Select(TC_Events.EtherCatEventClass.ErrorEvent)
		  	  .ArgSetSbRaise(sb.Set('Not linked EtherCAT master: ').AppendAny(ii));
		bChkEcHwLinked := FALSE;
		EXIT;
	END_IF
END_FOR

M_CheckEcHwLinked := bChkEcHwLinked;
END_METHOD

/// Function convert EtherCAT device state from a slave to ST_Text
METHOD PUBLIC M_ConvertEcDeviceStateToText : ST_Text
VAR_INPUT
	nDeviceState	: BYTE;
END_VAR
// switch EtherCAT device state
CASE nDeviceState OF
	/// init
	EC_DEVICE_STATE_INIT :
		M_ConvertEcDeviceStateToText := stTextListGlobal.stText_System.stText_EC_DeviceState_Init;
		
	/// preop
	EC_DEVICE_STATE_PREOP :
		M_ConvertEcDeviceStateToText := stTextListGlobal.stText_System.stText_EC_DeviceState_Preop;
	
	/// bootstrap
	EC_DEVICE_STATE_BOOTSTRAP :
		M_ConvertEcDeviceStateToText := stTextListGlobal.stText_System.stText_EC_DeviceState_Bootstrap;
	
	/// safeop
	EC_DEVICE_STATE_SAFEOP :
		M_ConvertEcDeviceStateToText := stTextListGlobal.stText_System.stText_EC_DeviceState_Safeop;
	
	/// op
	EC_DEVICE_STATE_OP :
		M_ConvertEcDeviceStateToText := stTextListGlobal.stText_System.stText_EC_DeviceState_Op;
	
	/// error
	EC_DEVICE_STATE_ERROR :
		M_ConvertEcDeviceStateToText := stTextListGlobal.stText_System.stText_EC_DeviceState_Error;
	
	/// invalid vprs
	EC_DEVICE_STATE_INVALID_VPRS :
		M_ConvertEcDeviceStateToText := stTextListGlobal.stText_System.stText_EC_DeviceState_InvalidVprs;
	
	/// init cmd error
	EC_DEVICE_STATE_INITCMD_ERROR :
		M_ConvertEcDeviceStateToText := stTextListGlobal.stText_System.stText_EC_DeviceState_InitCmdError;

	ELSE // default
		M_ConvertEcDeviceStateToText := stTextListGlobal.stText_System.stText_EC_DeviceState_Undefined;
	
END_CASE
END_METHOD

/// Function convert EtherCAT link state from a slave to ST_Text
METHOD PUBLIC M_ConvertEcLinkStateToText : ST_Text
VAR_INPUT
	nLinkState : BYTE;
END_VAR
// switch EtherCAT link state
CASE nLinkState OF
	/// ok
	EC_LINK_STATE_OK :
		M_ConvertEcLinkStateToText := stTextListGlobal.stText_System.stText_EC_LinkState_Ok;
		
	/// not present
	EC_LINK_STATE_NOT_PRESENT :
		M_ConvertEcLinkStateToText := stTextListGlobal.stText_System.stText_EC_LinkState_NotPresent;
	
	/// without com
	EC_LINK_STATE_LINK_WITHOUT_COMM :
		M_ConvertEcLinkStateToText := stTextListGlobal.stText_System.stText_EC_LinkState_WithoutCom;
	
	/// missing link
	EC_LINK_STATE_MISSING_LINK :
		M_ConvertEcLinkStateToText := stTextListGlobal.stText_System.stText_EC_LinkState_MissingLink;
	
	/// additional link
	EC_LINK_STATE_ADDITIONAL_LINK :
		M_ConvertEcLinkStateToText := stTextListGlobal.stText_System.stText_EC_LinkState_AdditionalLink;
	
	/// state port a
	EC_LINK_STATE_PORT_A :
		M_ConvertEcLinkStateToText := stTextListGlobal.stText_System.stText_EC_LinkState_PortA;
	
	/// state port b
	EC_LINK_STATE_PORT_B :
		M_ConvertEcLinkStateToText := stTextListGlobal.stText_System.stText_EC_LinkState_PortB;
	
	/// state port c
	EC_LINK_STATE_PORT_C :
		M_ConvertEcLinkStateToText := stTextListGlobal.stText_System.stText_EC_LinkState_PortC;
	
	/// state port d
	EC_LINK_STATE_PORT_D :
		M_ConvertEcLinkStateToText := stTextListGlobal.stText_System.stText_EC_LinkState_PortD;

	ELSE // default
		M_ConvertEcLinkStateToText := stTextListGlobal.stText_System.stText_EC_LinkState_Undefined;
	
END_CASE
END_METHOD

METHOD PUBLIC M_ConvertEcMasterStateToText : ST_Text
VAR_INPUT
	eEcState : E_EcDeviceState;
END_VAR
// switch EtherCAT master device state
CASE eEcState OF
	/// Link error
	eEtherCATState_LinkError :
		M_ConvertEcMasterStateToText := stTextListGlobal.stText_System.stText_EC_LinkError;
		
	/// I/O locked after link error (I/O reset required)
	eEtherCATState_IoLockedAfterLinkErr :
		M_ConvertEcMasterStateToText := stTextListGlobal.stText_System.stText_EC_IoLockedAfterLinkErr;
	
	/// Link error (redundancy adapter)
	eEtherCATState_LinkErrRedAdapter :
		M_ConvertEcMasterStateToText := stTextListGlobal.stText_System.stText_EC_LinkErrRedAdapter;
	
	/// Missing one frame (redundancy mode)
	eEtherCATState_MissingFrame :
		M_ConvertEcMasterStateToText := stTextListGlobal.stText_System.stText_EC_MissingFrame;
	
	/// Out of send resources (I/O reset required)
	eEtherCATState_OutOfSendResources :
		M_ConvertEcMasterStateToText := stTextListGlobal.stText_System.stText_EC_OutOfSendResources;
	
	/// Watchdog triggered
	eEtherCATState_WatchdogTriggered :
		M_ConvertEcMasterStateToText := stTextListGlobal.stText_System.stText_EC_WatchdogTriggered;
	
	/// Ethernet driver (miniport) not found
	eEtherCATState_EthernetDrvNotFound :
		M_ConvertEcMasterStateToText := stTextListGlobal.stText_System.stText_EC_EthernetDrvNotFound;
	
	/// I/O reset active
	eEtherCATState_IO_resetActive :
		M_ConvertEcMasterStateToText := stTextListGlobal.stText_System.stText_EC_IO_resetActive;
	
	/// At least one device in 'INIT' state
	eEtherCATState_AtLeastOneDeviceInit :
		M_ConvertEcMasterStateToText := stTextListGlobal.stText_System.stText_EC_AtLeastOneDeviceInit;
	
	///  At least one device in 'PRE-OP' state
	eEtherCATState_AtLeastOneDevicePreOp :
		M_ConvertEcMasterStateToText := stTextListGlobal.stText_System.stText_EC_AtLeastOneDevicePreOp;
	
	/// At least one device in 'SAFE-OP' state
	eEtherCATState_AtLeastOneDeviceSafeOp :
		M_ConvertEcMasterStateToText := stTextListGlobal.stText_System.stText_EC_AtLeastOneDeviceSafeOp;
	
	/// At least one device indicates an error state
	eEtherCATState_AtLeastOneDeviceError :
		M_ConvertEcMasterStateToText := stTextListGlobal.stText_System.stText_EC_AtLeastOneDeviceError;
	
	/// DC not in sync
	eEtherCATState_DC_notInSync :
		M_ConvertEcMasterStateToText := stTextListGlobal.stText_System.stText_EC_DC_notInSync;

	ELSE // default
		IF eEcState <> 0 THEN
			M_ConvertEcMasterStateToText := stTextListGlobal.stText_System.stText_EC_CommonError;
		ELSE
			M_ConvertEcMasterStateToText := stEmptyText;
		END_IF
	
END_CASE
END_METHOD

/// Dependency injection method.
{attribute 'object_name' := 'SetReferences'}
METHOD INTERNAL SetReferences
VAR_INPUT
	/// event access provider
	IEventHandler : I_EventHandler;
END_VAR
/// set up references
IEvent := IEventHandler;
END_METHOD

END_FUNCTION_BLOCK

// ---- POUs/System/P_SysSrv.TcPOU
PROGRAM P_SysSrv
VAR
	wsClearText				: WSTRING(255);		// clear text for debug
	
	fbShutDownHmi			: NT_StartProcess;
	fbStartAppEplan			: NT_StartProcess;
	fbStartAppCalculator	: NT_StartProcess;
	fbStartAppSetSystemTime	: NT_StartProcess;
	
	//    stSvcTime 		: TIMESTRUCT;
	//    wMsMir 			: WORD;
	//    fbNtSetTime 		: NT_SetLocalTime;
	//    diCntTimeSync		: UDINT;
	//    negSetTimeBusy	: F_TRIG;
END_VAR

// services
wsClearText := "Call fbEventHandler";
Services.fbEventHandler();

wsClearText := "Call fbRecipeManager";
Services.fbRecipeManager(
	stRecipe := Services.stSettings,
	nLogger := Services.ILog,
	bEnableLoadRecipe := stGlobalModuleInfo.bStation_All_Stopped, //stGlobalModuleInfo.bStation_All_InHome,
	fbVar2File := Services.fbVar2File);

wsClearText := "Call fbVar2File"; 
Services.fbVar2File(stConfig := stConfig.stVar2FileConfig);

// NT start process
fbShutDownHmi(
	NETID:= , 
	PATHSTR:= 'C:\Windows\System32\cmd.exe /C taskkill /F /IM msedge.exe', //Taskkill /F /IM Chrome.exe', 
	DIRNAME:= 'C:\Windows\System32' , 
	COMNDLINE:= , 
	START:= HMI.stHmi.stIn.stSpecial.stButton_CloseHmi.bClick, 
	TMOUT:= , 
	BUSY=> , 
	ERR=> , 
	ERRID=> );

fbStartAppCalculator(
	NETID:= , 
	PATHSTR:= 'C:\Windows\system32\calc.exe',//'C:\Windows\system32\win32calc.exe', 
	DIRNAME:= 'C:\Windows\system32',//'C:\Windows\system32', 
	COMNDLINE:= , 
	START:= HMI.stHmi.stIn.stSpecial.stButton_Calculator.bClick, 
	TMOUT:= , 
	BUSY=> , 
	ERR=> , 
	ERRID=> );

fbStartAppEplan(
	NETID:= , 
	PATHSTR:= 'C:\Windows\System32\cmd.exe /C\Tc3Apps\EPlan.pdf',
	DIRNAME:= 'C:\Windows\System32',
	COMNDLINE:= , 
	START:= HMI.stHmi.stIn.stSpecial.stButton_Eplan.bClick, 
	TMOUT:= , 
	BUSY=> , 
	ERR=> , 
	ERRID=> );	

fbStartAppSetSystemTime(
	NETID:= , 
	PATHSTR:='C:\Windows\System32\cmd.exe /C timedate.cpl', 
	DIRNAME:= 'C:\Windows\System32', 
	COMNDLINE:= , 
	START:= HMI.stHmi.stIn.stSpecial.stButton_SetSystemTime.bClick, 
	TMOUT:= , 
	BUSY=> , 
	ERR=> , 
	ERRID=> );

//// set up system time
//fbNtSetTime(
//                NETID:= '',
//                TIMESTR:= stSvcTime,
//                START:= stSvcTime.wMilliseconds <> wMsMir,
//                TMOUT:= ,
//                BUSY=> ,
//                ERR=> ,
//                ERRID=> );

//// rdy
//negSetTimeBusy(CLK := fbNtSetTime.BUSY);
//IF negSetTimeBusy.Q THEN
//                wMsMir := stSvcTime.wMilliseconds;
//                diCntTimeSync := diCntTimeSync + 1;
//END_IF

END_PROGRAM

// ---- Background/UnitTest/P_UnitTest.TcPOU
/// unit test program
PROGRAM P_UnitTest
VAR
	/// UnitTest VARs
	bInitDone			: BOOL;
	bRunTest			: BOOL := TRUE;
	bDone				: BOOL;
	bTestOk				: BOOL;
	ii					: INT;
	iStep				: INT;
	sLastError			: T_MaxString;
	IItem				: ITestCase;
	aTestItems			: ARRAY[0..iMaxIdxUnitTest] OF POINTER TO FB_TestCaseBase;
	/// test case instances
	fbTestFileLog		: FB_TestCase01FileLog;
	fbTestSystemInfo	: FB_TestCase02SystemInfo;
	fbTestStation		: FB_TestCase03Station;
	
END_VAR

///
/// Unit test program
///
/// TP www.rmth.at 2014
/// 
/// HOW TO
///		..run all tests:
/// 		simply set the bRunTest flag (overall test result --> bTestOk)
///
/// 	...add a test case:
///			1. copy a FB_TestCase... FB and rename it
///			2. implement test logic in Run method
///			3. add the instance in this Initialize method --> ready!
///	 

// call init action
IF NOT bInitDone THEN
	Initialize();
	RETURN;
END_IF

// call unit tests
CASE iStep OF
	0: 	// wait for start
		IF bRunTest THEN
			ii := 0;
			bDone := FALSE;
			bTestOk := TRUE;
			bRunTest := FALSE;
			sLastError := sEmpty;
			iStep := 10;	
		END_IF
		
	10:	// get next test case
		IF ii > iMaxIdxUnitTest THEN
			bDone := TRUE;
			iStep := 0;
		ELSIF aTestItems[ii] <> 0 THEN
			IItem := aTestItems[ii]^;
			iStep := 20;
		ELSE
			iStep := 50; 	// next test
		END_IF

	20:	// reset test item
		IItem.Reset();			
		IF IItem.TestState <> E_TestCaseState.eTestCaseState_ready OR IItem.TestResult <> E_TestResult.eTestResult_none THEN
			sLastError := Concat6('Test reset failed, test case index: ', INT_TO_STRING(ii), ' TestState: ', INT_TO_STRING(IItem.TestState), ' TestResult: ', INT_TO_STRING(IItem.TestResult));
			bTestOk := FALSE;
			iStep := 50; 	// next test 
		ELSE
			iStep := 30; 	// run test
		END_IF

	30:	// run test item
		IItem.Run();
		IF IItem.TestState <> E_TestCaseState.eTestCaseState_running THEN
			bTestOk := bTestOk AND IItem.TestState = E_TestCaseState.eTestCaseState_finished AND IItem.TestResult = E_TestResult.eTestResult_ok;
			IF IItem.TestState <> E_TestCaseState.eTestCaseState_finished OR IItem.TestResult <> E_TestResult.eTestResult_ok THEN
				sLastError := Concat6('Test failed, test case index: ', INT_TO_STRING(ii), ' TestState: ', INT_TO_STRING(IItem.TestState), ' TestResult: ', INT_TO_STRING(IItem.TestResult));
			END_IF
			iStep := 50; 	// next test
		END_IF
		
	50:	// next test item
		ii := ii + 1;
		iStep := 10;
END_CASE

